C05460=1018.869,-126.788,405.091,165.310,52.720,159.347
C05461=1018.864,-127.038,405.098,165.308,52.725,159.348
C05462=1018.858,-127.287,405.106,165.304,52.729,159.348
C05463=1018.854,-127.537,405.114,165.302,52.734,159.348
C05464=1018.848,-127.787,405.121,165.298,52.738,159.348
C05465=1018.843,-128.036,405.128,165.296,52.743,159.348
C05466=1018.839,-128.285,405.136,165.292,52.747,159.348
C05467=1018.834,-128.535,405.145,165.289,52.751,159.348
C05468=1018.830,-128.785,405.154,165.287,52.754,159.349
C05469=1018.827,-129.034,405.163,165.284,52.757,159.348
C05470=1018.824,-129.284,405.174,165.281,52.759,159.348
C05471=1018.821,-129.534,405.184,165.279,52.761,159.348
C05472=1018.819,-129.783,405.196,165.276,52.761,159.348
C05473=1018.817,-130.033,405.208,165.274,52.762,159.347
C05474=1018.816,-130.283,405.220,165.272,52.762,159.347
C05475=1018.815,-130.532,405.233,165.269,52.762,159.346
C05476=1018.815,-130.782,405.247,165.267,52.761,159.346
C05477=1018.815,-131.032,405.261,165.265,52.759,159.345
C05478=1018.815,-131.282,405.276,165.263,52.757,159.344
C05479=1018.816,-131.532,405.291,165.260,52.754,159.343
C05480=1018.817,-131.781,405.308,165.258,52.752,159.342
C05481=1018.819,-132.031,405.324,165.257,52.748,159.341
C05482=1018.821,-132.281,405.341,165.255,52.744,159.340
C05483=1018.823,-132.531,405.360,165.253,52.739,159.339
C05484=1018.827,-132.780,405.377,165.251,52.734,159.338
C05485=1018.830,-133.030,405.397,165.249,52.728,159.337
C05486=1018.834,-133.280,405.416,165.248,52.722,159.335
C05487=1018.565,-133.306,405.043,165.205,53.048,159.383
C05488=1018.561,-133.056,405.024,165.208,53.054,159.384
C05489=1018.558,-132.806,405.005,165.209,53.060,159.385
C05490=1018.554,-132.557,404.986,165.211,53.065,159.387
C05491=1018.552,-132.307,404.969,165.212,53.070,159.388
C05492=1018.550,-132.057,404.951,165.214,53.074,159.389
C05493=1018.549,-131.808,404.934,165.217,53.077,159.390
C05494=1018.547,-131.558,404.919,165.218,53.080,159.391
C05495=1018.546,-131.308,404.903,165.220,53.083,159.392
C05496=1018.546,-131.058,404.888,165.222,53.085,159.393
C05497=1018.546,-130.808,404.874,165.225,53.087,159.393
C05498=1018.547,-130.559,404.860,165.227,53.088,159.394
C05499=1018.547,-130.309,404.847,165.229,53.088,159.395
C05500=1018.549,-130.059,404.835,165.232,53.088,159.395
C05501=1018.550,-129.810,404.823,165.234,53.087,159.395
C05502=1018.552,-129.560,404.811,165.236,53.087,159.396
C05503=1018.555,-129.311,404.801,165.239,53.085,159.396
C05504=1018.558,-129.060,404.791,165.242,53.083,159.396
C05505=1018.562,-128.811,404.780,165.245,53.080,159.396
C05506=1018.566,-128.562,404.772,165.248,53.077,159.396
C05507=1018.569,-128.312,404.764,165.251,53.073,159.396
C05508=1018.574,-128.062,404.755,165.253,53.069,159.396
C05509=1018.580,-127.813,404.748,165.257,53.064,159.396
C05510=1018.584,-127.563,404.741,165.259,53.059,159.396
C05511=1018.590,-127.314,404.733,165.262,53.054,159.395
C05512=1018.595,-127.064,404.725,165.265,53.050,159.395
C05513=1018.600,-126.814,404.719,165.268,53.045,159.395
C05514=1018.605,-126.564,404.711,165.271,53.041,159.395
C05515=1018.611,-126.314,404.704,165.274,53.036,159.395
C05516=1018.615,-126.064,404.696,165.277,53.031,159.394
C05517=1018.621,-125.814,404.689,165.280,53.026,159.394
C05518=1018.625,-125.565,404.682,165.283,53.021,159.394
C05519=1018.631,-125.315,404.674,165.287,53.017,159.394
C05520=1018.636,-125.065,404.666,165.289,53.012,159.393
C05521=1018.641,-124.816,404.659,165.292,53.007,159.393
C05522=1018.646,-124.565,404.651,165.295,53.003,159.393
C05523=1018.652,-124.315,404.644,165.298,52.998,159.393
C05524=1018.656,-124.066,404.636,165.301,52.994,159.393
C05525=1018.661,-123.816,404.628,165.304,52.989,159.393
C05526=1018.667,-123.566,404.621,165.307,52.983,159.392
C05527=1018.672,-123.317,404.613,165.310,52.979,159.392
C05528=1018.677,-123.067,404.605,165.313,52.974,159.392
C05529=1018.682,-122.817,404.598,165.316,52.970,159.392
C05530=1018.687,-122.566,404.590,165.319,52.965,159.392
C05531=1018.692,-122.317,404.582,165.323,52.961,159.392
C05532=1018.698,-122.067,404.575,165.325,52.956,159.391
C05533=1018.703,-121.817,404.567,165.328,52.951,159.391
C05534=1018.707,-121.568,404.559,165.331,52.947,159.391
C05535=1018.713,-121.318,404.552,165.334,52.942,159.391
C05536=1018.718,-121.068,404.544,165.337,52.938,159.390
C05537=1018.723,-120.818,404.536,165.340,52.933,159.390
C05538=1018.728,-120.569,404.529,165.343,52.927,159.390
C05539=1018.734,-120.319,404.520,165.346,52.923,159.390
C05540=1018.739,-120.068,404.513,165.349,52.918,159.390
C05541=1018.744,-119.818,404.506,165.352,52.914,159.389
C05542=1018.749,-119.569,404.497,165.355,52.909,159.389
C05543=1018.754,-119.319,404.490,165.358,52.904,159.389
C05544=1018.759,-119.069,404.481,165.361,52.900,159.389
C05545=1018.765,-118.819,404.474,165.364,52.895,159.389
C05546=1018.770,-118.570,404.465,165.367,52.891,159.388
C05547=1018.774,-118.320,404.458,165.370,52.886,159.388
C05548=1018.781,-118.036,404.450,165.373,52.881,159.388
C05549=1018.786,-117.752,404.440,165.377,52.875,159.388
C05550=1018.793,-117.468,404.432,165.381,52.869,159.387
C05551=1018.798,-117.184,404.423,165.384,52.865,159.387
C05552=1018.804,-116.934,404.414,165.386,52.860,159.387
C05553=1018.809,-116.684,404.406,165.390,52.855,159.387
C05554=1018.814,-116.435,404.399,165.393,52.850,159.387
C05555=1018.819,-116.186,404.390,165.396,52.846,159.386
C05556=1018.824,-115.935,404.383,165.399,52.841,159.386
C05557=1018.830,-115.685,404.374,165.401,52.836,159.386
C05558=1018.835,-115.435,404.367,165.405,52.832,159.386
C05559=1018.841,-115.186,404.358,165.408,52.827,159.386
C05560=1018.846,-114.935,404.351,165.411,52.823,159.385
C05561=1018.850,-114.686,404.343,165.414,52.818,159.385
C05562=1018.855,-114.437,404.334,165.416,52.813,159.385
C05563=1018.861,-114.187,404.327,165.420,52.808,159.385
C05564=1018.866,-113.937,404.318,165.424,52.803,159.385
C05565=1018.872,-113.687,404.310,165.426,52.799,159.384
C05566=1018.877,-113.437,404.302,165.430,52.794,159.384
C05567=1018.882,-113.187,404.294,165.432,52.790,159.384
C05568=1018.887,-112.937,404.285,165.436,52.785,159.384
C05569=1018.892,-112.687,404.277,165.439,52.780,159.384
C05570=1018.897,-112.437,404.269,165.441,52.776,159.383
C05571=1018.902,-112.188,404.261,165.445,52.771,159.383
C05572=1018.908,-111.939,404.253,165.447,52.767,159.383
C05573=1018.913,-111.689,404.245,165.451,52.762,159.383
C05574=1018.918,-111.439,404.237,165.453,52.758,159.383
C05575=1018.924,-111.189,404.228,165.456,52.752,159.382
C05576=1018.929,-110.940,404.220,165.460,52.748,159.382
C05577=1018.934,-110.689,404.212,165.462,52.743,159.382
C05578=1018.939,-110.439,404.203,165.466,52.739,159.382
C05579=1018.944,-110.190,404.195,165.468,52.734,159.381
C05580=1018.950,-109.940,404.186,165.471,52.729,159.381
///RCONF 1,0,0,0,0,0,0,0,0,0,0,0,0,0,0,0,0,0,0,0,0,0,0,0
C05581=1018.955,-109.690,404.179,165.475,52.724,159.381
C05582=1018.961,-109.440,404.171,165.477,52.720,159.381
C05583=1018.966,-109.191,404.162,165.481,52.715,159.381
C05584=1018.971,-108.941,404.154,165.484,52.711,159.381
C05585=1018.976,-108.691,404.145,165.486,52.706,159.380
C05586=1018.982,-108.441,404.137,165.490,52.701,159.380
C05587=1018.987,-108.191,404.129,165.492,52.697,159.380
C05588=1018.992,-107.941,404.121,165.496,52.692,159.380
C05589=1018.997,-107.692,404.112,165.500,52.687,159.379
C05590=1019.002,-107.442,404.104,165.502,52.682,159.379
C05591=1019.008,-107.192,404.095,165.505,52.678,159.379
C05592=1019.013,-106.943,404.087,165.508,52.673,159.379
C05593=1019.018,-106.693,404.078,165.511,52.669,159.379
C05594=1019.023,-106.443,404.070,165.514,52.664,159.378
C05595=1019.029,-106.193,404.061,165.517,52.660,159.378
C05596=1019.035,-105.943,404.052,165.521,52.655,159.378
C05597=1019.040,-105.693,404.044,165.523,52.650,159.378
C05598=1019.045,-105.444,404.035,165.526,52.645,159.377
C05599=1019.050,-105.194,404.027,165.529,52.641,159.377
C05600=1019.056,-104.944,404.018,165.532,52.636,159.377
C05601=1019.060,-104.694,404.009,165.535,52.632,159.377
C05602=1019.065,-104.444,404.001,165.538,52.627,159.377
C05603=1019.071,-104.195,403.992,165.542,52.623,159.377
C05604=1019.076,-103.945,403.984,165.544,52.618,159.376
C05605=1019.081,-103.695,403.975,165.547,52.613,159.376
C05606=1019.087,-103.445,403.967,165.550,52.609,159.376
C05607=1019.092,-103.195,403.958,165.553,52.604,159.376
C05608=1019.098,-102.945,403.950,165.557,52.599,159.376
C05609=1019.103,-102.696,403.941,165.559,52.595,159.375
C05610=1019.108,-102.446,403.933,165.563,52.590,159.375
C05611=1019.113,-102.197,403.923,165.565,52.585,159.375
C05612=1019.119,-101.912,403.913,165.570,52.580,159.375
C05613=1019.125,-101.628,403.903,165.573,52.575,159.374
C05614=1019.131,-101.345,403.893,165.576,52.570,159.374
C05615=1019.138,-101.060,403.883,165.579,52.564,159.374
C05616=1019.143,-100.811,403.875,165.583,52.560,159.374
C05617=1019.148,-100.561,403.866,165.585,52.555,159.373
C05618=1019.153,-100.311,403.858,165.589,52.551,159.373
C05619=1019.159,-100.061,403.849,165.592,52.546,159.373
C05620=1019.164,-99.811,403.839,165.594,52.541,159.373
C05621=1019.169,-99.562,403.831,165.598,52.536,159.372
C05622=1019.175,-99.312,403.822,165.600,52.532,159.372
C05623=1019.180,-99.062,403.814,165.604,52.527,159.372
C05624=1019.186,-98.812,403.804,165.607,52.522,159.372
C05625=1019.191,-98.563,403.796,165.609,52.518,159.371
C05626=1019.197,-98.313,403.787,165.613,52.513,159.371
C05627=1019.202,-98.063,403.779,165.615,52.509,159.371
C05628=1019.207,-97.813,403.769,165.619,52.504,159.371
C05629=1019.213,-97.563,403.760,165.622,52.499,159.371
C05630=1019.218,-97.314,403.751,165.625,52.495,159.371
C05631=1019.223,-97.064,403.742,165.628,52.490,159.370
C05632=1019.229,-96.814,403.733,165.631,52.486,159.370
C05633=1019.233,-96.564,403.724,165.634,52.481,159.370
C05634=1019.239,-96.315,403.715,165.637,52.477,159.370
C05635=1019.244,-96.064,403.705,165.640,52.472,159.369
C05636=1019.249,-95.815,403.696,165.643,52.468,159.369
C05637=1019.255,-95.565,403.687,165.646,52.463,159.369
C05638=1019.259,-95.316,403.678,165.649,52.459,159.369
C05639=1019.265,-95.065,403.669,165.652,52.454,159.369
C05640=1019.270,-94.815,403.660,165.655,52.450,159.368
C05641=1019.275,-94.566,403.651,165.658,52.445,159.368
C05642=1019.281,-94.316,403.642,165.661,52.441,159.368
C05643=1019.286,-94.066,403.632,165.664,52.436,159.368
C05644=1019.291,-93.817,403.623,165.667,52.432,159.368
C05645=1019.297,-93.567,403.613,165.670,52.427,159.368
C05646=1019.302,-93.317,403.605,165.672,52.422,159.367
C05647=1019.308,-93.068,403.596,165.676,52.418,159.367
C05648=1019.313,-92.817,403.586,165.680,52.413,159.367
C05649=1019.318,-92.568,403.577,165.682,52.409,159.367
C05650=1019.323,-92.319,403.567,165.686,52.404,159.366
C05651=1019.329,-92.068,403.558,165.688,52.400,159.366
C05652=1019.334,-91.819,403.548,165.692,52.395,159.366
C05653=1019.339,-91.569,403.540,165.694,52.391,159.366
C05654=1019.345,-91.319,403.530,165.697,52.386,159.365
C05655=1019.350,-91.069,403.521,165.700,52.381,159.365
C05656=1019.356,-90.819,403.512,165.703,52.377,159.365
C05657=1019.361,-90.570,403.502,165.707,52.372,159.365
C05658=1019.366,-90.320,403.493,165.709,52.368,159.365
C05659=1019.372,-90.070,403.483,165.713,52.363,159.364
C05660=1019.377,-89.821,403.475,165.715,52.358,159.364
C05661=1019.383,-89.571,403.465,165.719,52.353,159.364
C05662=1019.388,-89.321,403.455,165.721,52.349,159.364
C05663=1019.394,-89.071,403.447,165.725,52.345,159.363
C05664=1019.399,-88.821,403.437,165.728,52.340,159.363
C05665=1019.405,-88.572,403.427,165.730,52.335,159.363
C05666=1019.409,-88.322,403.418,165.734,52.330,159.363
C05667=1019.415,-88.073,403.409,165.736,52.326,159.362
C05668=1019.420,-87.822,403.399,165.740,52.321,159.362
C05669=1019.425,-87.573,403.390,165.743,52.317,159.362
C05670=1019.432,-87.323,403.381,165.745,52.312,159.362
C05671=1019.436,-87.074,403.371,165.749,52.307,159.362
C05672=1019.443,-86.824,403.361,165.752,52.303,159.361
C05673=1019.447,-86.574,403.352,165.755,52.298,159.361
C05674=1019.453,-86.324,403.343,165.758,52.293,159.361
C05675=1019.458,-86.075,403.333,165.761,52.289,159.361
C05676=1019.465,-85.792,403.323,165.764,52.283,159.360
C05677=1019.471,-85.510,403.312,165.768,52.278,159.360
C05678=1019.477,-85.229,403.301,165.772,52.273,159.360
C05679=1019.483,-84.947,403.290,165.775,52.268,159.360
C05680=1019.489,-84.697,403.281,165.778,52.262,159.359
C05681=1019.494,-84.447,403.271,165.780,52.258,159.359
C05682=1019.500,-84.198,403.262,165.784,52.253,159.359
C05683=1019.505,-83.948,403.252,165.787,52.249,159.359
C05684=1019.511,-83.698,403.242,165.790,52.244,159.358
C05685=1019.516,-83.448,403.233,165.793,52.239,159.358
C05686=1019.522,-83.199,403.224,165.796,52.235,159.358
C05687=1019.528,-82.949,403.214,165.799,52.230,159.357
C05688=1019.533,-82.699,403.204,165.802,52.225,159.357
C05689=1019.539,-82.450,403.195,165.805,52.221,159.357
C05690=1019.544,-82.199,403.185,165.808,52.215,159.357
C05691=1019.550,-81.950,403.176,165.812,52.211,159.357
C05692=1019.555,-81.700,403.166,165.814,52.207,159.356
C05693=1019.561,-81.451,403.157,165.817,52.201,159.356
C05694=1019.566,-81.200,403.147,165.821,52.197,159.356
C05695=1019.572,-80.951,403.137,165.823,52.192,159.355
C05696=1019.577,-80.701,403.127,165.826,52.187,159.355
C05697=1019.583,-80.451,403.118,165.830,52.182,159.355
C05698=1019.589,-80.201,403.108,165.832,52.177,159.355
C05699=1019.594,-79.952,403.098,165.836,52.173,159.354
C05700=1019.600,-79.702,403.088,165.838,52.169,159.354
C05701=1019.605,-79.452,403.078,165.842,52.164,159.354
C05702=1019.610,-79.203,403.068,165.844,52.160,159.354
C05703=1019.616,-78.953,403.059,165.847,52.154,159.353
C05704=1019.621,-78.703,403.049,165.851,52.150,159.353
C05705=1019.626,-78.453,403.039,165.853,52.145,159.353
C05706=1019.632,-78.203,403.029,165.857,52.141,159.353
C05707=1019.638,-77.955,403.019,165.859,52.137,159.353
C05708=1019.643,-77.705,403.009,165.863,52.131,159.352
C05709=1019.648,-77.454,402.998,165.865,52.127,159.352
C05710=1019.654,-77.204,402.988,165.869,52.122,159.352
C05711=1019.659,-76.955,402.979,165.871,52.118,159.352
C05712=1019.665,-76.705,402.969,165.874,52.113,159.351
C05713=1019.670,-76.455,402.959,165.878,52.108,159.351
C05714=1019.675,-76.206,402.948,165.880,52.104,159.351
C05715=1019.682,-75.956,402.939,165.884,52.099,159.351
C05716=1019.687,-75.706,402.928,165.886,52.094,159.350
C05717=1019.693,-75.456,402.918,165.890,52.090,159.350
C05718=1019.697,-75.207,402.909,165.893,52.085,159.350
C05719=1019.704,-74.958,402.898,165.895,52.080,159.349
C05720=1019.709,-74.708,402.888,165.899,52.076,159.349
C05721=1019.715,-74.457,402.878,165.901,52.071,159.349
C05722=1019.720,-74.208,402.868,165.905,52.067,159.349
C05723=1019.725,-73.959,402.857,165.907,52.063,159.349
C05724=1019.731,-73.708,402.847,165.911,52.058,159.348
C05725=1019.736,-73.458,402.837,165.913,52.053,159.348
C05726=1019.741,-73.210,402.826,165.917,52.048,159.348
C05727=1019.747,-72.959,402.816,165.919,52.044,159.347
C05728=1019.752,-72.709,402.806,165.923,52.040,159.347
C05729=1019.758,-72.460,402.795,165.925,52.035,159.347
C05730=1019.763,-72.210,402.785,165.929,52.031,159.347
C05731=1019.768,-71.961,402.775,165.931,52.027,159.347
C05732=1019.774,-71.711,402.764,165.935,52.022,159.346
C05733=1019.780,-71.461,402.753,165.937,52.017,159.346
C05734=1019.785,-71.211,402.743,165.941,52.012,159.346
C05735=1019.790,-70.961,402.733,165.943,52.008,159.346
C05736=1019.796,-70.712,402.723,165.947,52.004,159.345
C05737=1019.800,-70.462,402.712,165.949,51.999,159.345
C05738=1019.806,-70.212,402.701,165.953,51.995,159.345
C05739=1019.812,-69.962,402.691,165.955,51.990,159.345
C05740=1019.818,-69.683,402.679,165.959,51.985,159.344
C05741=1019.824,-69.403,402.667,165.962,51.980,159.344
C05742=1019.830,-69.123,402.656,165.965,51.975,159.344
C05743=1019.837,-68.843,402.644,165.968,51.970,159.344
C05744=1019.842,-68.594,402.633,165.972,51.965,159.343
C05745=1019.847,-68.344,402.623,165.975,51.960,159.343
C05746=1019.853,-68.095,402.612,165.978,51.956,159.343
C05747=1019.858,-67.844,402.602,165.981,51.951,159.343
C05748=1019.864,-67.595,402.591,165.984,51.947,159.342
C05749=1019.869,-67.345,402.581,165.987,51.942,159.342
C05750=1019.875,-67.095,402.570,165.989,51.937,159.342
C05751=1019.880,-66.846,402.559,165.993,51.933,159.342
C05752=1019.886,-66.595,402.548,165.996,51.929,159.341
C05753=1019.891,-66.347,402.538,165.999,51.923,159.341
C05754=1019.896,-66.097,402.528,166.001,51.919,159.341
C05755=1019.902,-65.847,402.517,166.005,51.915,159.340
C05756=1019.908,-65.598,402.506,166.007,51.910,159.340
C05757=1019.913,-65.347,402.496,166.011,51.905,159.340
C05758=1019.919,-65.098,402.485,166.014,51.900,159.340
C05759=1019.925,-64.848,402.474,166.017,51.896,159.339
C05760=1019.930,-64.598,402.464,166.020,51.892,159.339
C05761=1019.936,-64.349,402.453,166.022,51.887,159.339
C05762=1019.941,-64.099,402.443,166.026,51.882,159.339
C05763=1019.947,-63.849,402.432,166.028,51.878,159.338
C05764=1019.952,-63.599,402.421,166.032,51.873,159.338
C05765=1019.958,-63.350,402.410,166.034,51.868,159.338
C05766=1019.963,-63.100,402.400,166.038,51.864,159.338
C05767=1019.969,-62.850,402.389,166.041,51.858,159.337
C05768=1019.975,-62.601,402.378,166.043,51.854,159.337
C05769=1019.980,-62.351,402.368,166.047,51.850,159.337
C05770=1019.986,-62.101,402.357,166.049,51.845,159.336
C05771=1019.991,-61.852,402.346,166.053,51.840,159.336
C05772=1019.997,-61.602,402.335,166.055,51.836,159.336
C05773=1020.003,-61.352,402.325,166.058,51.831,159.335
C05774=1020.008,-61.103,402.314,166.061,51.826,159.335
C05775=1020.013,-60.853,402.302,166.064,51.822,159.335
C05776=1020.019,-60.603,402.292,166.068,51.817,159.335
C05777=1020.025,-60.353,402.281,166.070,51.812,159.334
C05778=1020.030,-60.104,402.271,166.073,51.807,159.334
C05779=1020.036,-59.854,402.260,166.076,51.803,159.334
C05780=1020.042,-59.604,402.248,166.079,51.798,159.334
C05781=1020.048,-59.355,402.238,166.083,51.793,159.333
C05782=1020.054,-59.105,402.227,166.085,51.789,159.333
C05783=1020.059,-58.855,402.217,166.088,51.783,159.333
C05784=1020.065,-58.606,402.206,166.091,51.779,159.332
C05785=1020.070,-58.356,402.194,166.094,51.774,159.332
C05786=1020.076,-58.106,402.183,166.098,51.769,159.332
C05787=1020.082,-57.857,402.172,166.100,51.765,159.331
C05788=1020.087,-57.607,402.162,166.103,51.760,159.331
C05789=1020.093,-57.357,402.151,166.106,51.756,159.331
C05790=1020.099,-57.107,402.140,166.109,51.750,159.330
C05791=1020.105,-56.857,402.129,166.113,51.746,159.330
C05792=1020.110,-56.608,402.118,166.115,51.741,159.330
C05793=1020.116,-56.358,402.108,166.118,51.736,159.330
C05794=1020.121,-56.109,402.096,166.120,51.731,159.329
C05795=1020.127,-55.859,402.085,166.124,51.727,159.329
C05796=1020.133,-55.610,402.074,166.127,51.722,159.329
C05797=1020.139,-55.360,402.063,166.130,51.717,159.328
C05798=1020.144,-55.109,402.053,166.133,51.712,159.328
C05799=1020.150,-54.860,402.042,166.136,51.708,159.328
C05800=1020.156,-54.610,402.031,166.139,51.703,159.327
C05801=1020.162,-54.361,402.020,166.142,51.698,159.327
C05802=1020.167,-54.110,402.008,166.144,51.693,159.327
C05803=1020.173,-53.861,401.998,166.148,51.689,159.326
C05804=1020.180,-53.582,401.985,166.151,51.683,159.326
C05805=1020.186,-53.304,401.973,166.154,51.678,159.326
C05806=1020.193,-53.025,401.961,166.158,51.673,159.325
C05807=1020.199,-52.746,401.948,166.161,51.667,159.325
C05808=1020.205,-52.497,401.937,166.164,51.662,159.325
C05809=1020.211,-52.247,401.926,166.167,51.657,159.324
C05810=1020.216,-51.998,401.916,166.170,51.653,159.324
C05811=1020.223,-51.748,401.904,166.173,51.648,159.324
C05812=1020.228,-51.498,401.893,166.176,51.643,159.323
C05813=1020.233,-51.248,401.882,166.179,51.638,159.323
C05814=1020.239,-50.999,401.871,166.182,51.633,159.323
C05815=1020.245,-50.749,401.860,166.184,51.629,159.322
C05816=1020.251,-50.500,401.848,166.188,51.624,159.322
C05817=1020.257,-50.250,401.837,166.190,51.619,159.322
C05818=1020.262,-50.000,401.825,166.194,51.615,159.322
C05819=1020.268,-49.750,401.814,166.196,51.610,159.321
C05820=1020.273,-49.501,401.802,166.200,51.606,159.321
C05821=1020.279,-49.251,401.791,166.202,51.601,159.321
C05822=1020.285,-49.001,401.779,166.205,51.596,159.320
C05823=1020.290,-48.752,401.767,166.208,51.592,159.320
C05824=1020.296,-48.502,401.756,166.211,51.587,159.320
C05825=1020.301,-48.252,401.745,166.214,51.583,159.319
C05826=1020.307,-48.002,401.733,166.217,51.577,159.319
C05827=1020.312,-47.753,401.721,166.219,51.573,159.319
C05828=1020.318,-47.504,401.710,166.223,51.569,159.319
C05829=1020.324,-47.253,401.698,166.225,51.564,159.318
C05830=1020.330,-47.004,401.687,166.229,51.559,159.318
C05831=1020.335,-46.754,401.675,166.231,51.555,159.318
C05832=1020.341,-46.505,401.663,166.235,51.550,159.317
C05833=1020.346,-46.255,401.652,166.237,51.546,159.317
C05834=1020.352,-46.006,401.641,166.240,51.540,159.317
C05835=1020.358,-45.756,401.629,166.244,51.536,159.316
C05836=1020.364,-45.506,401.618,166.246,51.532,159.316
C05837=1020.369,-45.256,401.606,166.250,51.526,159.316
C05838=1020.375,-45.007,401.594,166.252,51.522,159.316
C05839=1020.380,-44.757,401.583,166.255,51.517,159.315
C05840=1020.386,-44.507,401.570,166.258,51.513,159.315
C05841=1020.392,-44.258,401.559,166.261,51.508,159.314
C05842=1020.397,-44.008,401.547,166.264,51.503,159.314
C05843=1020.404,-43.758,401.536,166.267,51.498,159.314
C05844=1020.409,-43.508,401.524,166.269,51.494,159.314
C05845=1020.415,-43.259,401.512,166.273,51.489,159.313
C05846=1020.420,-43.009,401.501,166.275,51.484,159.313
C05847=1020.426,-42.760,401.489,166.279,51.480,159.313
C05848=1020.432,-42.510,401.478,166.281,51.475,159.312
C05849=1020.437,-42.261,401.465,166.285,51.470,159.312
C05850=1020.444,-42.010,401.454,166.287,51.466,159.312
C05851=1020.449,-41.761,401.442,166.290,51.461,159.311
C05852=1020.455,-41.512,401.431,166.294,51.456,159.311
C05853=1020.460,-41.262,401.418,166.296,51.452,159.311
C05854=1020.466,-41.012,401.408,166.299,51.446,159.310
C05855=1020.472,-40.762,401.395,166.302,51.442,159.310
C05856=1020.478,-40.513,401.384,166.305,51.437,159.310
C05857=1020.484,-40.263,401.372,166.307,51.432,159.309
C05858=1020.489,-40.014,401.359,166.311,51.428,159.309
C05859=1020.495,-39.764,401.348,166.313,51.423,159.308
C05860=1020.501,-39.514,401.336,166.317,51.418,159.308
C05861=1020.507,-39.264,401.325,166.319,51.413,159.308
C05862=1020.512,-39.015,401.313,166.322,51.409,159.308
C05863=1020.518,-38.765,401.300,166.325,51.405,159.307
C05864=1020.523,-38.515,401.289,166.328,51.399,159.307
C05865=1020.529,-38.266,401.276,166.331,51.395,159.307
C05866=1020.535,-38.017,401.264,166.334,51.390,159.306
C05867=1020.541,-37.767,401.252,166.336,51.386,159.306
C05868=1020.547,-37.488,401.239,166.340,51.380,159.306
C05869=1020.553,-37.210,401.225,166.343,51.375,159.305
C05870=1020.559,-36.932,401.212,166.346,51.370,159.305
C05871=1020.566,-36.653,401.199,166.349,51.365,159.304
C05872=1020.572,-36.403,401.186,166.353,51.360,159.304
C05873=1020.577,-36.154,401.174,166.355,51.355,159.304
C05874=1020.583,-35.904,401.161,166.359,51.351,159.304
C05875=1020.588,-35.654,401.150,166.361,51.347,159.303
C05876=1020.595,-35.405,401.138,166.364,51.341,159.303
C05877=1020.600,-35.156,401.126,166.367,51.337,159.303
C05878=1020.606,-34.906,401.113,166.369,51.332,159.302
C05879=1020.612,-34.656,401.101,166.373,51.328,159.302
C05880=1020.617,-34.406,401.089,166.375,51.323,159.301
C05881=1020.623,-34.156,401.076,166.378,51.318,159.301
C05882=1020.629,-33.907,401.065,166.381,51.314,159.301
C05883=1020.635,-33.657,401.052,166.384,51.309,159.301
C05884=1020.640,-33.408,401.040,166.386,51.304,159.300
C05885=1020.646,-33.158,401.028,166.390,51.300,159.300
C05886=1020.652,-32.909,401.015,166.392,51.295,159.299
C05887=1020.657,-32.659,401.004,166.396,51.290,159.299
C05888=1020.663,-32.409,400.992,166.398,51.285,159.299
C05889=1020.669,-32.160,400.979,166.402,51.281,159.299
C05890=1020.675,-31.910,400.967,166.404,51.276,159.298
C05891=1020.681,-31.660,400.954,166.407,51.272,159.298
C05892=1020.686,-31.411,400.942,166.410,51.267,159.297
C05893=1020.692,-31.161,400.930,166.413,51.262,159.297
C05894=1020.698,-30.911,400.917,166.415,51.257,159.297
C05895=1020.704,-30.662,400.905,166.419,51.252,159.296
C05896=1020.710,-30.413,400.893,166.421,51.248,159.296
C05897=1020.716,-30.163,400.880,166.424,51.243,159.296
C05898=1020.721,-29.913,400.868,166.427,51.239,159.295
C05899=1020.727,-29.664,400.856,166.430,51.233,159.295
C05900=1020.733,-29.414,400.843,166.433,51.229,159.295
C05901=1020.738,-29.165,400.831,166.436,51.224,159.294
C05902=1020.745,-28.915,400.819,166.438,51.219,159.294
C05903=1020.751,-28.665,400.806,166.442,51.215,159.294
C05904=1020.756,-28.416,400.794,166.444,51.210,159.293
C05905=1020.762,-28.166,400.782,166.448,51.205,159.293
C05906=1020.768,-27.916,400.769,166.450,51.200,159.292
C05907=1020.774,-27.666,400.756,166.453,51.195,159.292
C05908=1020.779,-27.417,400.744,166.455,51.191,159.292
C05909=1020.785,-27.167,400.732,166.459,51.186,159.291
C05910=1020.791,-26.917,400.719,166.461,51.182,159.291
C05911=1020.797,-26.667,400.707,166.464,51.176,159.291
C05912=1020.802,-26.418,400.694,166.467,51.172,159.290
C05913=1020.808,-26.168,400.682,166.471,51.168,159.290
C05914=1020.813,-25.919,400.668,166.473,51.163,159.290
C05915=1020.819,-25.670,400.656,166.475,51.159,159.289
C05916=1020.825,-25.420,400.643,166.479,51.153,159.289
C05917=1020.830,-25.170,400.631,166.481,51.149,159.289
C05918=1020.836,-24.920,400.618,166.484,51.144,159.288
C05919=1020.842,-24.671,400.605,166.487,51.140,159.288
C05920=1020.848,-24.421,400.593,166.490,51.135,159.288
C05921=1020.853,-24.171,400.580,166.493,51.131,159.287
C05922=1020.859,-23.921,400.567,166.495,51.126,159.287
C05923=1020.865,-23.673,400.554,166.499,51.121,159.287
C05924=1020.870,-23.423,400.542,166.501,51.116,159.286
C05925=1020.876,-23.173,400.529,166.504,51.112,159.286
C05926=1020.882,-22.923,400.516,166.507,51.107,159.285
C05927=1020.889,-22.674,400.503,166.510,51.103,159.285
C05928=1020.893,-22.424,400.490,166.512,51.098,159.285
C05929=1020.899,-22.175,400.478,166.515,51.093,159.284
C05930=1020.905,-21.925,400.465,166.518,51.088,159.284
C05931=1020.911,-21.675,400.452,166.520,51.083,159.284
C05932=1020.918,-21.396,400.438,166.524,51.078,159.283
C05933=1020.924,-21.117,400.423,166.527,51.073,159.283
C05934=1020.930,-20.838,400.409,166.530,51.068,159.282
C05935=1020.936,-20.559,400.395,166.533,51.063,159.282
C05936=1020.942,-20.309,400.382,166.537,51.058,159.282
C05937=1020.948,-20.059,400.369,166.539,51.053,159.281
C05938=1020.954,-19.810,400.356,166.542,51.048,159.281
C05939=1020.961,-19.560,400.343,166.545,51.043,159.280
C05940=1020.967,-19.310,400.331,166.548,51.039,159.280
C05941=1020.971,-19.061,400.318,166.550,51.034,159.280
C05942=1020.977,-18.812,400.304,166.554,51.030,159.280
C05943=1020.983,-18.562,400.292,166.556,51.025,159.279
C05944=1020.989,-18.312,400.279,166.558,51.020,159.279
C05945=1020.995,-18.063,400.266,166.562,51.015,159.278
C05946=1021.001,-17.813,400.254,166.564,51.010,159.278
C05947=1021.007,-17.563,400.240,166.568,51.005,159.277
C05948=1021.013,-17.313,400.227,166.570,51.001,159.277
C05949=1021.019,-17.064,400.214,166.573,50.996,159.277
C05950=1021.024,-16.815,400.202,166.576,50.991,159.276
C05951=1021.030,-16.566,400.188,166.579,50.987,159.276
C05952=1021.036,-16.316,400.176,166.581,50.982,159.276
C05953=1021.041,-16.066,400.163,166.585,50.977,159.275
C05954=1021.048,-15.816,400.149,166.587,50.972,159.275
C05955=1021.054,-15.566,400.137,166.590,50.967,159.275
C05956=1021.059,-15.317,400.123,166.593,50.963,159.274
C05957=1021.065,-15.068,400.110,166.595,50.958,159.274
C05958=1021.070,-14.817,400.097,166.598,50.953,159.273
C05959=1021.077,-14.568,400.083,166.601,50.949,159.273
C05960=1021.083,-14.319,400.070,166.603,50.944,159.272
C05961=1021.088,-14.069,400.057,166.607,50.940,159.272
C05962=1021.094,-13.819,400.044,166.609,50.935,159.272
C05963=1021.099,-13.569,400.031,166.613,50.930,159.272
C05964=1021.106,-13.320,400.017,166.615,50.926,159.271
C05965=1021.111,-13.070,400.003,166.618,50.921,159.271
C05966=1021.116,-12.821,399.991,166.621,50.916,159.270
C05967=1021.123,-12.572,399.978,166.623,50.912,159.270
C05968=1021.128,-12.322,399.964,166.627,50.907,159.270
C05969=1021.134,-12.073,399.951,166.629,50.902,159.269
C05970=1021.139,-11.823,399.938,166.631,50.898,159.269
C05971=1021.146,-11.574,399.924,166.635,50.893,159.268
C05972=1021.151,-11.324,399.910,166.637,50.889,159.268
C05973=1021.157,-11.074,399.898,166.640,50.883,159.268
C05974=1021.163,-10.825,399.884,166.643,50.879,159.267
C05975=1021.169,-10.575,399.871,166.645,50.875,159.267
C05976=1021.175,-10.326,399.858,166.649,50.869,159.267
C05977=1021.180,-10.076,399.844,166.651,50.865,159.266
C05978=1021.186,-9.827,399.831,166.654,50.860,159.266
C05979=1021.192,-9.577,399.817,166.657,50.855,159.265
C05980=1021.199,-9.327,399.804,166.659,50.850,159.265
C05981=1021.204,-9.077,399.790,166.662,50.846,159.265
C05982=1021.210,-8.828,399.777,166.665,50.841,159.264
C05983=1021.216,-8.578,399.763,166.668,50.836,159.264
C05984=1021.222,-8.329,399.750,166.671,50.832,159.263
C05985=1021.227,-8.079,399.736,166.674,50.827,159.263
C05986=1021.233,-7.829,399.724,166.676,50.822,159.263
C05987=1021.239,-7.580,399.710,166.679,50.818,159.262
C05988=1021.245,-7.330,399.697,166.682,50.813,159.262
C05989=1021.251,-7.081,399.683,166.684,50.808,159.261
C05990=1021.257,-6.832,399.669,166.688,50.803,159.261
C05991=1021.262,-6.582,399.657,166.690,50.798,159.261
C05992=1021.268,-6.332,399.643,166.693,50.793,159.260
C05993=1021.274,-6.083,399.630,166.695,50.788,159.260
C05994=1021.280,-5.833,399.615,166.698,50.784,159.259
C05995=1021.286,-5.583,399.602,166.701,50.779,159.259
C05996=1021.293,-5.303,399.587,166.704,50.774,159.259
C05997=1021.299,-5.021,399.572,166.707,50.768,159.258
C05998=1021.306,-4.741,399.556,166.711,50.763,159.258
C05999=1021.312,-4.459,399.541,166.714,50.758,159.257
C06000=1021.318,-4.210,399.528,166.716,50.753,159.257
C06001=1021.324,-3.960,399.514,166.719,50.748,159.256
C06002=1021.329,-3.711,399.500,166.722,50.744,159.256
C06003=1021.336,-3.461,399.487,166.724,50.739,159.255
C06004=1021.342,-3.211,399.473,166.727,50.735,159.255
C06005=1021.348,-2.962,399.458,166.730,50.730,159.255
C06006=1021.353,-2.713,399.444,166.733,50.726,159.254
C06007=1021.358,-2.463,399.431,166.735,50.721,159.254
C06008=1021.364,-2.213,399.417,166.739,50.716,159.254
C06009=1021.370,-1.964,399.403,166.741,50.711,159.253
C06010=1021.376,-1.714,399.389,166.743,50.707,159.253
C06011=1021.382,-1.464,399.375,166.747,50.702,159.253
C06012=1021.387,-1.215,399.362,166.749,50.697,159.252
C06013=1021.393,-0.966,399.347,166.751,50.693,159.252
C06014=1021.398,-0.716,399.333,166.755,50.688,159.251
C06015=1021.405,-0.467,399.320,166.757,50.683,159.251
C06016=1021.411,-0.217,399.306,166.760,50.679,159.250
C06017=1021.416,0.033,399.292,166.763,50.674,159.250
C06018=1021.422,0.282,399.278,166.765,50.670,159.250
C06019=1021.427,0.531,399.263,166.768,50.665,159.249
C06020=1021.434,0.781,399.250,166.771,50.660,159.249
C06021=1021.439,1.030,399.236,166.774,50.656,159.249
C06022=1021.445,1.281,399.222,166.776,50.651,159.248
C06023=1021.451,1.530,399.208,166.779,50.646,159.248
C06024=1021.457,1.779,399.193,166.782,50.642,159.247
C06025=1021.462,2.029,399.180,166.784,50.637,159.247
C06026=1021.468,2.279,399.165,166.788,50.633,159.247
C06027=1021.474,2.528,399.152,166.790,50.628,159.246
C06028=1021.480,2.778,399.138,166.792,50.623,159.246
C06029=1021.486,3.027,399.124,166.796,50.619,159.245
C06030=1021.492,3.277,399.109,166.798,50.614,159.245
C06031=1021.497,3.527,399.096,166.800,50.609,159.244
C06032=1021.503,3.776,399.081,166.803,50.604,159.244
C06033=1021.509,4.025,399.068,166.806,50.600,159.244
C06034=1021.515,4.275,399.053,166.809,50.595,159.243
C06035=1021.521,4.525,399.040,166.811,50.590,159.243
C06036=1021.526,4.774,399.025,166.814,50.586,159.242
C06037=1021.532,5.023,399.011,166.817,50.581,159.242
C06038=1021.538,5.273,398.997,166.820,50.576,159.241
C06039=1021.544,5.522,398.983,166.822,50.571,159.241
C06040=1021.550,5.772,398.969,166.826,50.567,159.241
C06041=1021.556,6.022,398.955,166.828,50.562,159.240
C06042=1021.562,6.271,398.940,166.830,50.557,159.240
C06043=1021.567,6.520,398.926,166.833,50.552,159.239
C06044=1021.573,6.770,398.913,166.836,50.548,159.239
C06045=1021.579,7.020,398.898,166.838,50.543,159.238
C06046=1021.585,7.269,398.884,166.841,50.538,159.238
C06047=1021.591,7.519,398.870,166.844,50.533,159.238
C06048=1021.597,7.768,398.856,166.847,50.529,159.237
C06049=1021.603,8.018,398.842,166.850,50.524,159.237
C06050=1021.608,8.267,398.827,166.852,50.519,159.236
C06051=1021.615,8.517,398.813,166.855,50.514,159.236
C06052=1021.620,8.767,398.799,166.857,50.509,159.235
C06053=1021.627,9.016,398.785,166.860,50.505,159.235
C06054=1021.633,9.266,398.771,166.863,50.500,159.235
C06055=1021.638,9.514,398.756,166.865,50.495,159.234
C06056=1021.644,9.781,398.741,166.869,50.490,159.234
C06057=1021.651,10.048,398.726,166.872,50.485,159.233
C06058=1021.658,10.314,398.711,166.874,50.479,159.233
C06059=1021.664,10.580,398.695,166.877,50.474,159.232
C06060=1021.670,10.845,398.680,166.880,50.469,159.232
C06061=1021.676,11.112,398.665,166.883,50.464,159.231
C06062=1021.683,11.378,398.650,166.886,50.459,159.231
C06063=1021.689,11.644,398.635,166.889,50.454,159.231
C06064=1021.695,11.893,398.620,166.891,50.449,159.230
C06065=1021.701,12.144,398.606,166.894,50.445,159.229
C06066=1021.707,12.393,398.591,166.897,50.439,159.229
C06067=1021.713,12.643,398.577,166.899,50.435,159.229
C06068=1021.719,12.892,398.563,166.903,50.429,159.228
C06069=1021.725,13.142,398.548,166.905,50.425,159.228
C06070=1021.731,13.391,398.534,166.907,50.420,159.227
C06071=1021.736,13.641,398.520,166.911,50.416,159.227
C06072=1021.743,13.890,398.505,166.913,50.411,159.226
C06073=1021.748,14.139,398.490,166.915,50.406,159.226
C06074=1021.754,14.390,398.476,166.919,50.401,159.225
C06075=1021.760,14.638,398.462,166.921,50.397,159.225
C06076=1021.767,14.888,398.447,166.923,50.392,159.225
C06077=1021.771,15.138,398.432,166.927,50.387,159.224
C06078=1021.777,15.387,398.418,166.929,50.382,159.224
C06079=1021.784,15.637,398.403,166.932,50.378,159.223
C06080=1021.789,15.886,398.389,166.935,50.373,159.223
C06081=1021.795,16.136,398.374,166.937,50.368,159.222
C06082=1021.801,16.385,398.359,166.939,50.363,159.222
C06083=1021.807,16.635,398.344,166.943,50.359,159.222
C06084=1021.812,16.884,398.330,166.945,50.354,159.221
C06085=1021.819,17.134,398.315,166.948,50.349,159.221
C06086=1021.824,17.383,398.300,166.951,50.344,159.220
C06087=1021.831,17.633,398.285,166.953,50.340,159.220
C06088=1021.836,17.882,398.272,166.956,50.335,159.219
C06089=1021.843,18.132,398.257,166.958,50.331,159.219
C06090=1021.848,18.381,398.241,166.961,50.326,159.219
C06091=1021.854,18.631,398.227,166.964,50.321,159.218
C06092=1021.860,18.880,398.213,166.966,50.316,159.217
C06093=1021.866,19.130,398.198,166.969,50.311,159.217
C06094=1021.872,19.379,398.183,166.972,50.307,159.217
C06095=1021.877,19.629,398.168,166.974,50.302,159.216
C06096=1021.883,19.878,398.153,166.977,50.297,159.216
C06097=1021.890,20.128,398.138,166.980,50.292,159.215
C06098=1021.894,20.377,398.124,166.982,50.288,159.215
C06099=1021.901,20.627,398.109,166.986,50.283,159.215
C06100=1021.906,20.876,398.094,166.988,50.278,159.214
C06101=1021.912,21.126,398.079,166.990,50.274,159.214
C06102=1021.918,21.375,398.064,166.992,50.269,159.213
C06103=1021.924,21.625,398.049,166.996,50.264,159.213
C06104=1021.931,21.874,398.034,166.998,50.260,159.212
C06105=1021.936,22.124,398.019,167.001,50.255,159.212
C06106=1021.942,22.373,398.004,167.004,50.250,159.211
C06107=1021.948,22.622,397.989,167.006,50.245,159.211
C06108=1021.954,22.872,397.974,167.009,50.241,159.211
C06109=1021.959,23.121,397.959,167.012,50.236,159.210
C06110=1021.966,23.371,397.944,167.014,50.231,159.210
C06111=1021.971,23.621,397.929,167.017,50.226,159.209
C06112=1021.977,23.870,397.914,167.019,50.222,159.209
C06113=1021.984,24.119,397.899,167.022,50.216,159.208
C06114=1021.989,24.369,397.884,167.025,50.212,159.208
C06115=1021.995,24.618,397.869,167.027,50.208,159.207
C06116=1022.001,24.868,397.854,167.030,50.203,159.207
C06117=1022.006,25.117,397.839,167.033,50.198,159.206
C06118=1022.013,25.367,397.824,167.035,50.193,159.206
C06119=1022.019,25.616,397.809,167.038,50.188,159.205
C06120=1022.024,25.866,397.794,167.040,50.183,159.205
C06121=1022.031,26.115,397.779,167.043,50.179,159.205
C06122=1022.036,26.364,397.764,167.046,50.174,159.204
C06123=1022.042,26.614,397.749,167.049,50.169,159.204
C06124=1022.049,26.899,397.732,167.052,50.164,159.203
C06125=1022.055,27.183,397.715,167.055,50.158,159.203
C06126=1022.062,27.467,397.697,167.058,50.153,159.202
C06127=1022.069,27.752,397.680,167.061,50.148,159.202
C06128=1022.074,28.001,397.665,167.063,50.143,159.201
C06129=1022.081,28.251,397.650,167.066,50.138,159.201
C06130=1022.086,28.501,397.634,167.068,50.133,159.200
C06131=1022.092,28.749,397.620,167.072,50.129,159.200
C06132=1022.098,28.999,397.603,167.074,50.124,159.199
C06133=1022.104,29.248,397.589,167.076,50.119,159.199
C06134=1022.109,29.498,397.573,167.079,50.115,159.198
C06135=1022.115,29.748,397.558,167.082,50.110,159.198
C06136=1022.122,29.997,397.542,167.085,50.106,159.198
C06137=1022.127,30.246,397.527,167.087,50.101,159.197
C06138=1022.133,30.496,397.512,167.089,50.096,159.196
C06139=1022.139,30.746,397.496,167.092,50.091,159.196
C06140=1022.145,30.994,397.481,167.095,50.086,159.196
C06141=1022.151,31.244,397.466,167.097,50.082,159.195
C06142=1022.156,31.494,397.450,167.101,50.077,159.195
C06143=1022.162,31.743,397.436,167.103,50.072,159.194
C06144=1022.168,31.992,397.419,167.105,50.068,159.194
C06145=1022.174,32.242,397.404,167.108,50.063,159.193
C06146=1022.180,32.492,397.389,167.111,50.058,159.193
C06147=1022.186,32.740,397.373,167.113,50.053,159.192
C06148=1022.192,32.990,397.358,167.115,50.048,159.192
C06149=1022.197,33.240,397.342,167.118,50.044,159.191
C06150=1022.203,33.489,397.328,167.121,50.039,159.191
C06151=1022.209,33.738,397.312,167.124,50.035,159.190
C06152=1022.215,33.988,397.297,167.126,50.030,159.190
C06153=1022.221,34.238,397.281,167.129,50.025,159.190
C06154=1022.227,34.486,397.266,167.132,50.020,159.189
C06155=1022.233,34.736,397.250,167.134,50.015,159.189
C06156=1022.239,34.986,397.234,167.137,50.010,159.188
C06157=1022.245,35.235,397.219,167.139,50.005,159.188
C06158=1022.250,35.485,397.204,167.142,50.001,159.187
C06159=1022.257,35.734,397.188,167.144,49.996,159.187
C06160=1022.262,35.984,397.173,167.147,49.991,159.186
C06161=1022.268,36.234,397.157,167.150,49.987,159.186
C06162=1022.275,36.483,397.141,167.152,49.982,159.185
C06163=1022.280,36.732,397.126,167.156,49.977,159.185
C06164=1022.286,36.981,397.110,167.158,49.972,159.184
C06165=1022.292,37.231,397.095,167.160,49.968,159.184
C06166=1022.298,37.480,397.079,167.163,49.963,159.183
C06167=1022.304,37.730,397.063,167.166,49.958,159.183
C06168=1022.309,37.979,397.047,167.169,49.954,159.183
C06169=1022.315,38.229,397.032,167.171,49.949,159.182
C06170=1022.321,38.478,397.016,167.173,49.944,159.181
C06171=1022.327,38.728,397.001,167.176,49.939,159.181
C06172=1022.333,38.977,396.984,167.179,49.935,159.181
C06173=1022.338,39.226,396.969,167.181,49.930,159.180
C06174=1022.344,39.476,396.953,167.184,49.926,159.180
C06175=1022.350,39.725,396.937,167.186,49.921,159.179
C06176=1022.356,39.975,396.921,167.189,49.916,159.179
C06177=1022.362,40.224,396.905,167.192,49.911,159.178
C06178=1022.368,40.474,396.890,167.194,49.907,159.178
C06179=1022.373,40.723,396.874,167.196,49.902,159.177
C06180=1022.379,40.972,396.858,167.200,49.897,159.177
C06181=1022.385,41.222,396.842,167.202,49.892,159.176
C06182=1022.391,41.471,396.826,167.205,49.888,159.176
C06183=1022.397,41.721,396.811,167.208,49.883,159.175
C06184=1022.403,41.970,396.795,167.210,49.878,159.175
C06185=1022.409,42.219,396.779,167.212,49.874,159.174
C06186=1022.414,42.469,396.763,167.215,49.869,159.174
C06187=1022.420,42.718,396.747,167.218,49.864,159.173
C06188=1022.427,43.003,396.728,167.220,49.859,159.173
C06189=1022.433,43.287,396.711,167.223,49.853,159.172
C06190=1022.440,43.571,396.693,167.227,49.848,159.172
C06191=1022.447,43.855,396.674,167.230,49.843,159.171
C06192=1022.453,44.105,396.658,167.232,49.839,159.171
C06193=1022.458,44.354,396.641,167.235,49.834,159.170
C06194=1022.463,44.604,396.625,167.237,49.829,159.170
C06195=1022.469,44.854,396.609,167.240,49.825,159.170
C06196=1022.475,45.102,396.593,167.242,49.820,159.169
C06197=1022.481,45.352,396.577,167.245,49.815,159.169
C06198=1022.487,45.601,396.561,167.248,49.811,159.168
C06199=1022.493,45.850,396.544,167.250,49.806,159.168
C06200=1022.498,46.100,396.529,167.253,49.802,159.167
C06201=1022.503,46.350,396.512,167.255,49.797,159.167
C06202=1022.509,46.599,396.496,167.258,49.792,159.166
C06203=1022.515,46.849,396.479,167.261,49.787,159.166
C06204=1022.521,47.098,396.463,167.263,49.783,159.165
C06205=1022.527,47.348,396.447,167.266,49.779,159.165
C06206=1022.533,47.596,396.431,167.268,49.774,159.164
C06207=1022.538,47.846,396.416,167.271,49.769,159.164
C06208=1022.544,48.095,396.399,167.274,49.764,159.163
C06209=1022.549,48.345,396.382,167.276,49.760,159.163
C06210=1022.555,48.594,396.366,167.278,49.755,159.162
C06211=1022.561,48.844,396.350,167.280,49.750,159.162
C06212=1022.567,49.093,396.334,167.284,49.746,159.162
C06213=1022.573,49.343,396.317,167.286,49.741,159.161
C06214=1022.579,49.592,396.301,167.289,49.736,159.161
C06215=1022.585,49.841,396.285,167.291,49.732,159.160
C06216=1022.591,50.091,396.269,167.294,49.727,159.160
C06217=1022.596,50.340,396.252,167.297,49.722,159.159
C06218=1022.602,50.590,396.236,167.299,49.717,159.159
C06219=1022.608,50.839,396.219,167.301,49.713,159.158
C06220=1022.614,51.088,396.203,167.305,49.708,159.158
C06221=1022.620,51.338,396.187,167.307,49.704,159.157
C06222=1022.626,51.587,396.170,167.310,49.699,159.157
C06223=1022.632,51.836,396.154,167.312,49.694,159.156
C06224=1022.637,52.086,396.137,167.314,49.689,159.156
C06225=1022.643,52.335,396.121,167.318,49.684,159.155
C06226=1022.649,52.585,396.105,167.320,49.680,159.155
C06227=1022.655,52.834,396.089,167.322,49.675,159.154
C06228=1022.661,53.083,396.072,167.325,49.670,159.154
C06229=1022.667,53.333,396.056,167.328,49.665,159.153
C06230=1022.673,53.582,396.040,167.330,49.661,159.153
C06231=1022.678,53.832,396.023,167.333,49.656,159.152
C06232=1022.684,54.081,396.007,167.335,49.651,159.152
C06233=1022.690,54.330,395.990,167.338,49.646,159.151
C06234=1022.696,54.580,395.974,167.341,49.641,159.151
C06235=1022.702,54.829,395.958,167.343,49.637,159.150
C06236=1022.708,55.078,395.942,167.346,49.633,159.150
C06237=1022.714,55.328,395.925,167.349,49.628,159.149
C06238=1022.719,55.577,395.909,167.351,49.623,159.149
C06239=1022.725,55.827,395.892,167.354,49.618,159.148
C06240=1022.731,56.076,395.876,167.357,49.613,159.148
C06241=1022.737,56.326,395.859,167.359,49.609,159.147
C06242=1022.744,56.575,395.842,167.362,49.604,159.147
C06243=1022.750,56.824,395.826,167.364,49.599,159.146
C06244=1022.755,57.074,395.809,167.367,49.594,159.146
C06245=1022.761,57.323,395.793,167.370,49.590,159.145
C06246=1022.767,57.573,395.777,167.372,49.585,159.145
C06247=1022.773,57.822,395.761,167.374,49.580,159.144
C06248=1022.779,58.071,395.744,167.377,49.575,159.144
C06249=1022.785,58.320,395.727,167.380,49.570,159.143
C06250=1022.791,58.569,395.711,167.382,49.565,159.143
C06251=1022.797,58.820,395.694,167.386,49.560,159.142
C06252=1022.803,59.104,395.675,167.388,49.555,159.142
C06253=1022.810,59.388,395.657,167.391,49.550,159.141
C06254=1022.817,59.671,395.638,167.394,49.544,159.140
C06255=1022.824,59.956,395.619,167.397,49.538,159.140
C06256=1022.830,60.205,395.603,167.399,49.534,159.139
C06257=1022.836,60.454,395.586,167.403,49.529,159.139
C06258=1022.842,60.704,395.569,167.405,49.524,159.138
C06259=1022.848,60.953,395.553,167.407,49.519,159.138
C06260=1022.854,61.203,395.536,167.411,49.514,159.137
C06261=1022.860,61.452,395.520,167.413,49.510,159.137
C06262=1022.866,61.701,395.503,167.415,49.505,159.136
C06263=1022.872,61.950,395.487,167.419,49.500,159.136
C06264=1022.878,62.201,395.470,167.421,49.495,159.135
C06265=1022.884,62.450,395.453,167.423,49.490,159.135
C06266=1022.890,62.699,395.436,167.425,49.485,159.134
C06267=1022.896,62.948,395.420,167.429,49.480,159.134
C06268=1022.902,63.197,395.404,167.431,49.476,159.133
C06269=1022.908,63.447,395.386,167.433,49.471,159.133
C06270=1022.914,63.696,395.370,167.437,49.466,159.132
C06271=1022.919,63.946,395.353,167.439,49.461,159.132
C06272=1022.925,64.195,395.336,167.441,49.457,159.131
C06273=1022.931,64.444,395.319,167.444,49.452,159.131
C06274=1022.937,64.694,395.302,167.446,49.447,159.130
C06275=1022.943,64.944,395.285,167.449,49.442,159.130
C06276=1022.949,65.193,395.269,167.452,49.438,159.129
C06277=1022.954,65.442,395.251,167.454,49.433,159.129
C06278=1022.960,65.691,395.235,167.457,49.428,159.128
C06279=1022.966,65.941,395.217,167.460,49.423,159.128
C06280=1022.972,66.190,395.201,167.462,49.419,159.127
C06281=1022.978,66.439,395.183,167.465,49.414,159.127
C06282=1022.984,66.689,395.167,167.467,49.409,159.126
C06283=1022.990,66.939,395.149,167.471,49.405,159.126
C06284=1022.996,67.188,395.133,167.473,49.400,159.125
C06285=1023.001,67.437,395.115,167.475,49.396,159.125
C06286=1023.007,67.686,395.099,167.478,49.391,159.124
C06287=1023.013,67.935,395.081,167.481,49.386,159.124
C06288=1023.019,68.185,395.065,167.483,49.381,159.123
C06289=1023.025,68.434,395.047,167.486,49.377,159.123
C06290=1023.030,68.683,395.029,167.488,49.372,159.122
C06291=1023.036,68.933,395.013,167.491,49.367,159.122
C06292=1023.042,69.183,394.995,167.494,49.362,159.121
C06293=1023.048,69.432,394.978,167.496,49.358,159.121
C06294=1023.054,69.681,394.961,167.499,49.353,159.120
C06295=1023.059,69.930,394.944,167.501,49.348,159.120
C06296=1023.065,70.180,394.927,167.504,49.343,159.119
C06297=1023.071,70.429,394.910,167.507,49.339,159.119
C06298=1023.077,70.678,394.892,167.509,49.334,159.118
C06299=1023.082,70.928,394.875,167.511,49.329,159.118
C06300=1023.089,71.177,394.858,167.514,49.325,159.117
C06301=1023.094,71.426,394.840,167.517,49.320,159.117
C06302=1023.100,71.676,394.823,167.519,49.315,159.116
C06303=1023.107,71.925,394.806,167.522,49.310,159.116
C06304=1023.112,72.174,394.789,167.524,49.306,159.115
C06305=1023.117,72.424,394.772,167.528,49.301,159.115
C06306=1023.123,72.673,394.754,167.530,49.297,159.114
C06307=1023.130,72.922,394.737,167.533,49.292,159.114
C06308=1023.135,73.172,394.719,167.535,49.288,159.113
C06309=1023.140,73.421,394.702,167.537,49.283,159.113
C06310=1023.147,73.671,394.685,167.541,49.278,159.112
C06311=1023.153,73.920,394.667,167.543,49.273,159.112
C06312=1023.158,74.169,394.650,167.545,49.269,159.111
C06313=1023.164,74.419,394.633,167.548,49.264,159.111
C06314=1023.170,74.668,394.616,167.551,49.259,159.110
C06315=1023.176,74.917,394.598,167.554,49.254,159.110
C06316=1023.183,75.201,394.578,167.557,49.249,159.109
C06317=1023.189,75.485,394.559,167.560,49.243,159.108
C06318=1023.196,75.769,394.539,167.562,49.238,159.108
C06319=1023.203,76.053,394.519,167.565,49.233,159.107
C06320=1023.208,76.302,394.501,167.568,49.228,159.107
C06321=1023.215,76.551,394.484,167.571,49.223,159.106
C06322=1023.221,76.801,394.466,167.573,49.219,159.106
C06323=1023.226,77.050,394.450,167.576,49.214,159.105
C06324=1023.231,77.299,394.432,167.578,49.209,159.105
C06325=1023.238,77.549,394.414,167.581,49.204,159.104
C06326=1023.243,77.798,394.396,167.584,49.200,159.104
C06327=1023.249,78.048,394.379,167.586,49.195,159.103
C06328=1023.255,78.297,394.361,167.588,49.190,159.103
C06329=1023.260,78.546,394.343,167.591,49.186,159.102
C06330=1023.266,78.796,394.325,167.595,49.181,159.102
C06331=1023.272,79.045,394.308,167.597,49.177,159.101
C06332=1023.277,79.294,394.290,167.599,49.172,159.101
C06333=1023.284,79.543,394.272,167.602,49.168,159.100
C06334=1023.289,79.793,394.255,167.604,49.163,159.100
C06335=1023.295,80.042,394.237,167.607,49.158,159.099
C06336=1023.301,80.291,394.219,167.610,49.153,159.099
C06337=1023.306,80.540,394.202,167.612,49.149,159.098
C06338=1023.312,80.790,394.184,167.615,49.144,159.098
C06339=1023.318,81.039,394.166,167.617,49.139,159.097
C06340=1023.324,81.289,394.148,167.620,49.134,159.097
C06341=1023.330,81.538,394.131,167.623,49.130,159.096
C06342=1023.335,81.787,394.113,167.625,49.125,159.096
C06343=1023.341,82.037,394.095,167.628,49.121,159.095
C06344=1023.347,82.286,394.078,167.631,49.116,159.095
C06345=1023.353,82.535,394.060,167.634,49.112,159.094
C06346=1023.359,82.784,394.042,167.636,49.107,159.094
C06347=1023.365,83.034,394.024,167.638,49.102,159.093
C06348=1023.370,83.283,394.006,167.641,49.098,159.093
C06349=1023.376,83.532,393.988,167.644,49.093,159.092
C06350=1023.382,83.781,393.971,167.647,49.088,159.092
C06351=1023.387,84.030,393.953,167.649,49.084,159.091
C06352=1023.394,84.280,393.935,167.651,49.079,159.091
C06353=1023.399,84.529,393.917,167.655,49.074,159.090
C06354=1023.405,84.779,393.900,167.657,49.069,159.090
C06355=1023.411,85.027,393.881,167.659,49.065,159.089
C06356=1023.417,85.277,393.863,167.662,49.060,159.089
C06357=1023.423,85.526,393.846,167.665,49.055,159.088
C06358=1023.429,85.776,393.828,167.668,49.051,159.088
C06359=1023.434,86.025,393.810,167.670,49.046,159.087
C06360=1023.440,86.275,393.792,167.672,49.041,159.087
C06361=1023.446,86.524,393.775,167.676,49.036,159.086
C06362=1023.452,86.773,393.756,167.678,49.032,159.086
C06363=1023.458,87.022,393.739,167.681,49.027,159.085
C06364=1023.464,87.272,393.721,167.684,49.022,159.085
C06365=1023.469,87.521,393.703,167.686,49.018,159.084
C06366=1023.476,87.770,393.685,167.689,49.013,159.084
C06367=1023.481,88.019,393.667,167.691,49.008,159.083
C06368=1023.488,88.269,393.649,167.694,49.003,159.082
C06369=1023.493,88.518,393.631,167.697,48.998,159.082
C06370=1023.499,88.767,393.613,167.699,48.994,159.081
C06371=1023.505,89.016,393.595,167.701,48.989,159.081
C06372=1023.511,89.266,393.577,167.705,48.984,159.080
C06373=1023.517,89.516,393.559,167.707,48.979,159.080
C06374=1023.522,89.765,393.541,167.710,48.975,159.079
C06375=1023.528,90.014,393.522,167.712,48.971,159.079
C06376=1023.533,90.263,393.504,167.716,48.966,159.078
C06377=1023.540,90.512,393.486,167.718,48.961,159.078
C06378=1023.545,90.761,393.468,167.721,48.957,159.077
C06379=1023.551,91.011,393.450,167.723,48.952,159.077
C06380=1023.557,91.295,393.429,167.726,48.946,159.076
C06381=1023.564,91.579,393.408,167.729,48.942,159.076
C06382=1023.571,91.863,393.387,167.732,48.936,159.075
C06383=1023.577,92.146,393.367,167.735,48.931,159.075
C06384=1023.583,92.396,393.348,167.738,48.926,159.074
C06385=1023.588,92.645,393.330,167.741,48.922,159.074
C06386=1023.595,92.894,393.311,167.743,48.917,159.073
C06387=1023.599,93.143,393.293,167.745,48.913,159.073
C06388=1023.606,93.392,393.275,167.749,48.908,159.072
C06389=1023.612,93.642,393.257,167.751,48.903,159.072
C06390=1023.617,93.891,393.238,167.754,48.898,159.071
C06391=1023.623,94.141,393.220,167.756,48.894,159.071
C06392=1023.629,94.389,393.202,167.760,48.889,159.070
C06393=1023.634,94.639,393.183,167.762,48.884,159.070
C06394=1023.641,94.888,393.164,167.764,48.880,159.069
C06395=1023.646,95.137,393.147,167.767,48.875,159.068
C06396=1023.652,95.387,393.128,167.770,48.870,159.068
C06397=1023.658,95.636,393.110,167.773,48.866,159.067
C06398=1023.664,95.885,393.091,167.775,48.861,159.067
C06399=1023.669,96.135,393.073,167.777,48.856,159.066
C06400=1023.675,96.383,393.055,167.781,48.851,159.066
C06401=1023.681,96.633,393.037,167.783,48.847,159.065
C06402=1023.687,96.883,393.017,167.786,48.842,159.065
C06403=1023.692,97.132,393.000,167.788,48.838,159.064
C06404=1023.699,97.381,392.981,167.791,48.833,159.064
C06405=1023.705,97.630,392.962,167.794,48.828,159.063
C06406=1023.710,97.879,392.944,167.796,48.824,159.063
C06407=1023.717,98.128,392.926,167.800,48.819,159.062
C06408=1023.722,98.378,392.907,167.802,48.814,159.062
C06409=1023.728,98.627,392.889,167.804,48.809,159.061
C06410=1023.734,98.876,392.870,167.807,48.805,159.061
C06411=1023.740,99.126,392.852,167.810,48.800,159.060
C06412=1023.745,99.374,392.833,167.813,48.795,159.060
C06413=1023.751,99.624,392.815,167.815,48.791,159.059
C06414=1023.757,99.874,392.796,167.818,48.786,159.059
C06415=1023.762,100.122,392.777,167.821,48.781,159.058
C06416=1023.768,100.372,392.758,167.824,48.777,159.058
C06417=1023.774,100.621,392.740,167.826,48.773,159.057
C06418=1023.779,100.870,392.721,167.829,48.768,159.057
C06419=1023.786,101.119,392.703,167.832,48.763,159.056
C06420=1023.791,101.369,392.683,167.834,48.759,159.056
C06421=1023.797,101.618,392.664,167.837,48.754,159.055
C06422=1023.802,101.867,392.647,167.839,48.750,159.055
C06423=1023.808,102.117,392.627,167.843,48.745,159.054
C06424=1023.814,102.366,392.608,167.845,48.740,159.054
C06425=1023.820,102.615,392.590,167.848,48.736,159.053
C06426=1023.825,102.864,392.571,167.850,48.732,159.053
C06427=1023.831,103.114,392.552,167.854,48.727,159.052
C06428=1023.837,103.362,392.534,167.856,48.722,159.052
C06429=1023.842,103.612,392.515,167.858,48.718,159.051
C06430=1023.849,103.861,392.496,167.861,48.713,159.051
C06431=1023.854,104.110,392.477,167.864,48.708,159.050
C06432=1023.859,104.359,392.458,167.867,48.703,159.050
C06433=1023.866,104.608,392.439,167.869,48.699,159.049
C06434=1023.871,104.858,392.421,167.872,48.694,159.049
C06435=1023.877,105.108,392.401,167.875,48.689,159.048
C06436=1023.883,105.356,392.383,167.877,48.685,159.048
C06437=1023.888,105.606,392.364,167.880,48.680,159.047
C06438=1023.894,105.855,392.345,167.882,48.676,159.047
C06439=1023.901,106.104,392.326,167.886,48.671,159.046
C06440=1023.906,106.353,392.307,167.888,48.667,159.046
C06441=1023.911,106.602,392.288,167.891,48.662,159.045
C06442=1023.918,106.851,392.269,167.894,48.657,159.045
C06443=1023.923,107.101,392.250,167.897,48.653,159.044
C06444=1023.930,107.385,392.229,167.900,48.647,159.044
C06445=1023.937,107.669,392.207,167.903,48.642,159.043
C06446=1023.943,107.953,392.186,167.906,48.637,159.043
C06447=1023.950,108.237,392.164,167.908,48.632,159.042
C06448=1023.956,108.486,392.145,167.912,48.627,159.041
C06449=1023.961,108.735,392.126,167.914,48.622,159.041
C06450=1023.967,108.984,392.107,167.917,48.618,159.040
C06451=1023.973,109.233,392.088,167.920,48.613,159.040
C06452=1023.979,109.483,392.069,167.923,48.608,159.039
C06453=1023.985,109.732,392.050,167.925,48.604,159.039
C06454=1023.991,109.981,392.031,167.929,48.599,159.038
C06455=1023.996,110.230,392.012,167.931,48.594,159.038
C06456=1024.002,110.480,391.993,167.933,48.590,159.037
C06457=1024.007,110.729,391.973,167.936,48.585,159.037
C06458=1024.014,110.978,391.955,167.940,48.581,159.036
C06459=1024.019,111.228,391.936,167.942,48.576,159.036
C06460=1024.025,111.477,391.916,167.944,48.572,159.035
C06461=1024.030,111.726,391.897,167.948,48.567,159.035
C06462=1024.036,111.975,391.878,167.950,48.562,159.034
C06463=1024.043,112.224,391.859,167.953,48.558,159.034
C06464=1024.048,112.473,391.840,167.956,48.553,159.033
C06465=1024.054,112.723,391.820,167.959,48.548,159.033
C06466=1024.060,112.972,391.801,167.961,48.544,159.032
C06467=1024.065,113.222,391.781,167.964,48.540,159.032
C06468=1024.070,113.470,391.762,167.966,48.535,159.031
C06469=1024.076,113.719,391.742,167.970,48.530,159.031
C06470=1024.081,113.969,391.723,167.972,48.526,159.030
C06471=1024.087,114.218,391.703,167.975,48.522,159.030
C06472=1024.093,114.467,391.684,167.977,48.517,159.029
C06473=1024.099,114.716,391.665,167.981,48.513,159.029
C06474=1024.105,114.966,391.646,167.983,48.508,159.028
C06475=1024.110,115.214,391.626,167.986,48.503,159.028
C06476=1024.115,115.464,391.606,167.988,48.500,159.028
C06477=1024.121,115.713,391.587,167.992,48.495,159.027
C06478=1024.127,115.962,391.567,167.994,48.490,159.027
C06479=1024.132,116.211,391.548,167.997,48.486,159.026
C06480=1024.138,116.460,391.528,167.999,48.481,159.025
C06481=1024.144,116.710,391.508,168.003,48.477,159.025
C06482=1024.150,116.959,391.489,168.005,48.472,159.025
C06483=1024.155,117.207,391.470,168.008,48.468,159.024
C06484=1024.160,117.457,391.450,168.011,48.463,159.024
C06485=1024.166,117.706,391.431,168.014,48.458,159.023
C06486=1024.172,117.955,391.411,168.017,48.454,159.023
C06487=1024.177,118.205,391.391,168.019,48.450,159.022
C06488=1024.183,118.453,391.371,168.022,48.445,159.022
C06489=1024.189,118.703,391.352,168.025,48.441,159.021
C06490=1024.195,118.952,391.333,168.027,48.436,159.021
C06491=1024.201,119.201,391.313,168.031,48.431,159.020
C06492=1024.206,119.451,391.293,168.034,48.427,159.020
C06493=1024.212,119.700,391.273,168.036,48.423,159.019
C06494=1024.217,119.949,391.254,168.038,48.418,159.019
C06495=1024.223,120.198,391.234,168.042,48.413,159.018
C06496=1024.229,120.447,391.215,168.044,48.409,159.018
C06497=1024.235,120.696,391.195,168.047,48.404,159.017
C06498=1024.241,120.946,391.175,168.050,48.399,159.017
C06499=1024.246,121.195,391.155,168.053,48.395,159.016
C06500=1024.252,121.444,391.136,168.056,48.391,159.016
C06501=1024.258,121.693,391.116,168.059,48.386,159.015
C06502=1024.263,121.942,391.096,168.061,48.382,159.015
C06503=1024.269,122.191,391.077,168.064,48.377,159.014
C06504=1024.275,122.441,391.057,168.067,48.372,159.014
C06505=1024.281,122.689,391.037,168.070,48.368,159.013
C06506=1024.286,122.939,391.017,168.072,48.363,159.013
C06507=1024.292,123.188,390.998,168.076,48.359,159.012
C06508=1024.298,123.472,390.975,168.079,48.353,159.012
C06509=1024.305,123.755,390.953,168.082,48.348,159.011
C06510=1024.312,124.039,390.931,168.086,48.343,159.011
C06511=1024.319,124.323,390.908,168.089,48.338,159.010
C06512=1024.324,124.573,390.889,168.091,48.333,159.010
C06513=1024.330,124.822,390.868,168.094,48.329,159.009
C06514=1024.336,125.071,390.848,168.098,48.324,159.009
C06515=1024.341,125.320,390.829,168.100,48.320,159.008
C06516=1024.347,125.569,390.809,168.103,48.315,159.008
C06517=1024.353,125.818,390.790,168.106,48.310,159.007
C06518=1024.359,126.067,390.770,168.109,48.306,159.007
C06519=1024.364,126.316,390.749,168.112,48.301,159.006
C06520=1024.370,126.566,390.730,168.114,48.297,159.006
C06521=1024.376,126.815,390.710,168.117,48.292,159.005
C06522=1024.382,127.063,390.690,168.120,48.287,159.005
C06523=1024.388,127.313,390.671,168.123,48.283,159.004
C06524=1024.394,127.562,390.650,168.126,48.279,159.004
C06525=1024.399,127.811,390.630,168.129,48.274,159.003
C06526=1024.405,128.061,390.611,168.132,48.269,159.003
C06527=1024.411,128.310,390.591,168.135,48.265,159.002
C06528=1024.417,128.558,390.571,168.137,48.260,159.002
C06529=1024.423,128.808,390.551,168.140,48.256,159.001
C06530=1024.429,129.057,390.532,168.143,48.251,159.001
C06531=1024.434,129.306,390.511,168.146,48.246,159.000
C06532=1024.441,129.555,390.491,168.149,48.241,159.000
C06533=1024.446,129.805,390.471,168.152,48.237,158.999
C06534=1024.452,130.054,390.451,168.155,48.232,158.999
C06535=1024.458,130.302,390.431,168.158,48.228,158.998
C06536=1024.464,130.552,390.411,168.161,48.224,158.998
C06537=1024.470,130.800,390.391,168.164,48.219,158.997
C06538=1024.475,131.050,390.371,168.167,48.214,158.997
C06539=1024.481,131.299,390.351,168.169,48.210,158.996
C06540=1024.486,131.549,390.330,168.173,48.206,158.996
C06541=1024.492,131.798,390.310,168.175,48.201,158.995
C06542=1024.498,132.047,390.290,168.178,48.197,158.995
C06543=1024.504,132.295,390.270,168.181,48.192,158.994
C06544=1024.509,132.545,390.249,168.184,48.188,158.994
C06545=1024.515,132.793,390.229,168.187,48.183,158.993
C06546=1024.520,133.043,390.209,168.190,48.179,158.993
C06547=1024.527,133.292,390.188,168.192,48.174,158.992
C06548=1024.532,133.541,390.168,168.196,48.169,158.992
C06549=1024.538,133.790,390.148,168.199,48.166,158.992
C06550=1024.543,134.039,390.127,168.201,48.161,158.991
C06551=1024.549,134.288,390.107,168.205,48.156,158.991
C06552=1024.555,134.538,390.086,168.207,48.152,158.990
C06553=1024.561,134.787,390.066,168.211,48.148,158.990
C06554=1024.566,135.036,390.046,168.213,48.143,158.989
C06555=1024.572,135.284,390.026,168.216,48.139,158.989
C06556=1024.578,135.534,390.005,168.219,48.134,158.988
C06557=1024.584,135.783,389.985,168.222,48.129,158.988
C06558=1024.589,136.032,389.965,168.226,48.125,158.987
C06559=1024.595,136.281,389.944,168.228,48.121,158.987
C06560=1024.601,136.530,389.924,168.231,48.116,158.986
C06561=1024.606,136.779,389.903,168.234,48.111,158.986
C06562=1024.613,137.029,389.883,168.237,48.108,158.985
C06563=1024.618,137.278,389.863,168.240,48.103,158.985
C06564=1024.623,137.527,389.842,168.243,48.098,158.984
C06565=1024.629,137.775,389.821,168.245,48.094,158.984
C06566=1024.635,138.025,389.800,168.249,48.089,158.983
C06567=1024.641,138.274,389.780,168.252,48.085,158.983
C06568=1024.646,138.523,389.760,168.255,48.080,158.982
C06569=1024.652,138.772,389.739,168.258,48.076,158.982
C06570=1024.658,139.022,389.718,168.260,48.072,158.982
C06571=1024.664,139.270,389.698,168.264,48.067,158.981
C06572=1024.670,139.554,389.675,168.267,48.062,158.981
C06573=1024.676,139.838,389.651,168.271,48.057,158.980
C06574=1024.683,140.122,389.627,168.274,48.052,158.980
C06575=1024.689,140.406,389.603,168.278,48.047,158.979
C06576=1024.695,140.655,389.583,168.280,48.043,158.979
C06577=1024.701,140.904,389.563,168.284,48.038,158.978
C06578=1024.707,141.153,389.541,168.286,48.034,158.978
C06579=1024.712,141.402,389.521,168.290,48.029,158.977
C06580=1024.717,141.651,389.500,168.292,48.025,158.977
C06581=1024.724,141.901,389.480,168.295,48.020,158.976
C06582=1024.729,142.149,389.458,168.299,48.016,158.976
C06583=1024.735,142.398,389.438,168.301,48.012,158.975
C06584=1024.740,142.647,389.417,168.305,48.007,158.975
C06585=1024.746,142.896,389.396,168.307,48.003,158.974
C06586=1024.752,143.145,389.376,168.311,47.998,158.974
C06587=1024.757,143.394,389.355,168.313,47.994,158.973
C06588=1024.763,143.644,389.333,168.316,47.990,158.973
C06589=1024.769,143.893,389.313,168.320,47.985,158.973
C06590=1024.775,144.141,389.292,168.322,47.981,158.972
C06591=1024.781,144.391,389.271,168.326,47.976,158.972
C06592=1024.786,144.640,389.251,168.328,47.972,158.971
C06593=1024.792,144.889,389.229,168.332,47.968,158.971
C06594=1024.798,145.138,389.209,168.334,47.963,158.970
C06595=1024.804,145.386,389.188,168.338,47.959,158.970
C06596=1024.810,145.636,389.167,168.341,47.954,158.969
C06597=1024.815,145.885,389.146,168.344,47.950,158.969
C06598=1024.820,146.134,389.125,168.347,47.945,158.968
C06599=1024.826,146.384,389.104,168.351,47.941,158.968
C06600=1024.832,146.632,389.083,168.353,47.937,158.967
C06601=1024.838,146.882,389.062,168.356,47.933,158.967
C06602=1024.843,147.131,389.041,168.359,47.928,158.967
C06603=1024.849,147.379,389.020,168.362,47.924,158.966
C06604=1024.855,147.629,388.999,168.366,47.919,158.966
C06605=1024.860,147.877,388.977,168.368,47.915,158.965
C06606=1024.866,148.127,388.956,168.372,47.910,158.965
C06607=1024.872,148.376,388.935,168.375,47.906,158.964
C06608=1024.877,148.625,388.915,168.378,47.902,158.964
C06609=1024.883,148.874,388.893,168.381,47.898,158.963
C06610=1024.889,149.123,388.872,168.384,47.893,158.963
C06611=1024.895,149.372,388.851,168.387,47.889,158.962
C06612=1024.900,149.621,388.829,168.390,47.885,158.962
C06613=1024.906,149.869,388.808,168.393,47.880,158.962
C06614=1024.912,150.119,388.787,168.396,47.876,158.961
C06615=1024.917,150.368,388.766,168.400,47.871,158.961
C06616=1024.923,150.617,388.744,168.402,47.867,158.960
C06617=1024.929,150.866,388.724,168.406,47.863,158.960
C06618=1024.935,151.115,388.702,168.408,47.858,158.959
C06619=1024.940,151.364,388.681,168.412,47.854,158.959
C06620=1024.946,151.614,388.660,168.415,47.850,158.958
C06621=1024.952,151.862,388.639,168.418,47.845,158.958
C06622=1024.957,152.111,388.617,168.421,47.841,158.958
C06623=1024.963,152.360,388.596,168.425,47.837,158.957
C06624=1024.969,152.609,388.575,168.427,47.833,158.957
C06625=1024.975,152.858,388.554,168.431,47.828,158.956
C06626=1024.980,153.107,388.532,168.433,47.824,158.956
C06627=1024.986,153.356,388.510,168.437,47.819,158.955
C06628=1024.991,153.605,388.490,168.440,47.815,158.955
C06629=1024.997,153.854,388.468,168.444,47.811,158.955
C06630=1025.003,154.103,388.447,168.446,47.806,158.954
C06631=1025.009,154.352,388.425,168.450,47.802,158.954
C06632=1025.014,154.601,388.403,168.452,47.798,158.953
C06633=1025.020,154.850,388.382,168.456,47.794,158.953
C06634=1025.025,155.099,388.361,168.459,47.789,158.952
C06635=1025.031,155.348,388.339,168.463,47.785,158.952
C06636=1025.038,155.632,388.314,168.466,47.780,158.951
C06637=1025.044,155.915,388.290,168.469,47.775,158.951
C06638=1025.051,156.199,388.266,168.473,47.770,158.950
C06639=1025.058,156.482,388.241,168.476,47.766,158.950
C06640=1025.063,156.731,388.219,168.480,47.761,158.950
C06641=1025.069,156.980,388.197,168.484,47.757,158.949
C06642=1025.074,157.229,388.176,168.486,47.752,158.949
C06643=1025.081,157.478,388.155,168.490,47.748,158.948
C06644=1025.085,157.727,388.133,168.493,47.744,158.948
C06645=1025.091,157.976,388.111,168.496,47.740,158.947
C06646=1025.097,158.225,388.090,168.499,47.735,158.947
C06647=1025.103,158.474,388.068,168.503,47.731,158.947
C06648=1025.109,158.724,388.047,168.505,47.727,158.946
C06649=1025.114,158.973,388.025,168.509,47.722,158.946
C06650=1025.120,159.221,388.003,168.512,47.718,158.945
C06651=1025.125,159.470,387.981,168.515,47.714,158.945
C06652=1025.131,159.719,387.960,168.518,47.710,158.944
C06653=1025.137,159.969,387.937,168.522,47.706,158.944
C06654=1025.142,160.217,387.915,168.525,47.702,158.944
C06655=1025.148,160.467,387.894,168.528,47.697,158.943
C06656=1025.153,160.715,387.871,168.531,47.693,158.943
C06657=1025.158,160.964,387.849,168.535,47.689,158.943
C06658=1025.164,161.213,387.828,168.538,47.686,158.942
C06659=1025.169,161.462,387.805,168.541,47.681,158.942
C06660=1025.175,161.711,387.783,168.544,47.677,158.941
C06661=1025.181,161.960,387.761,168.548,47.673,158.941
C06662=1025.186,162.209,387.739,168.550,47.669,158.940
C06663=1025.191,162.458,387.716,168.554,47.664,158.940
C06664=1025.197,162.707,387.695,168.557,47.661,158.940
C06665=1025.203,162.956,387.673,168.561,47.656,158.939
C06666=1025.208,163.205,387.651,168.563,47.652,158.939
C06667=1025.214,163.454,387.628,168.567,47.648,158.939
C06668=1025.219,163.702,387.607,168.570,47.644,158.938
C06669=1025.224,163.952,387.584,168.574,47.640,158.938
C06670=1025.231,164.201,387.562,168.576,47.636,158.937
C06671=1025.236,164.449,387.540,168.580,47.632,158.937
C06672=1025.241,164.699,387.518,168.583,47.627,158.936
C06673=1025.247,164.947,387.496,168.587,47.623,158.936
C06674=1025.252,165.196,387.474,168.590,47.619,158.936
C06675=1025.258,165.445,387.451,168.593,47.615,158.935
C06676=1025.263,165.695,387.428,168.597,47.611,158.935
C06677=1025.269,165.943,387.407,168.600,47.607,158.935
C06678=1025.275,166.192,387.384,168.603,47.602,158.934
C06679=1025.280,166.442,387.362,168.606,47.599,158.934
C06680=1025.286,166.689,387.340,168.610,47.594,158.933
C06681=1025.291,166.939,387.318,168.612,47.590,158.933
C06682=1025.297,167.188,387.295,168.616,47.586,158.933
C06683=1025.303,167.437,387.273,168.620,47.582,158.932
C06684=1025.308,167.686,387.251,168.623,47.577,158.932
C06685=1025.314,167.935,387.228,168.626,47.573,158.931
C06686=1025.320,168.184,387.207,168.629,47.570,158.931
C06687=1025.326,168.433,387.184,168.633,47.566,158.931
C06688=1025.331,168.682,387.162,168.637,47.561,158.930
C06689=1025.336,168.931,387.139,168.640,47.557,158.930
C06690=1025.343,169.180,387.117,168.643,47.553,158.930
C06691=1025.348,169.429,387.094,168.646,47.549,158.929
C06692=1025.353,169.677,387.072,168.650,47.545,158.929
C06693=1025.360,169.926,387.050,168.654,47.541,158.928
C06694=1025.365,170.175,387.027,168.656,47.536,158.928
C06695=1025.371,170.425,387.005,168.660,47.532,158.927
C06696=1025.376,170.673,386.982,168.664,47.528,158.927
C06697=1025.382,170.922,386.961,168.667,47.524,158.927
C06698=1025.388,171.171,386.938,168.670,47.520,158.926
C06699=1025.393,171.420,386.915,168.674,47.516,158.926
C06700=1025.400,171.703,386.890,168.678,47.511,158.926
C06701=1025.406,171.986,386.865,168.681,47.506,158.925
C06702=1025.413,172.269,386.839,168.685,47.502,158.925
C06703=1025.419,172.552,386.813,168.689,47.497,158.924
C06704=1025.426,172.801,386.791,168.692,47.493,158.924
C06705=1025.431,173.051,386.769,168.696,47.489,158.923
C06706=1025.436,173.299,386.746,168.700,47.484,158.923
C06707=1025.442,173.548,386.723,168.702,47.480,158.923
C06708=1025.448,173.797,386.701,168.706,47.476,158.922
C06709=1025.454,174.046,386.679,168.710,47.472,158.922
C06710=1025.460,174.295,386.656,168.714,47.468,158.921
C06711=1025.466,174.544,386.634,168.716,47.464,158.921
C06712=1025.472,174.793,386.611,168.720,47.460,158.921
C06713=1025.477,175.042,386.588,168.724,47.455,158.920
C06714=1025.483,175.291,386.565,168.727,47.451,158.920
C06715=1025.489,175.539,386.544,168.731,47.447,158.920
C06716=1025.494,175.788,386.521,168.734,47.443,158.919
C06717=1025.500,176.037,386.498,168.738,47.439,158.919
C06718=1025.506,176.286,386.475,168.741,47.435,158.918
C06719=1025.512,176.535,386.453,168.745,47.431,158.918
C06720=1025.518,176.784,386.430,168.748,47.426,158.918
C06721=1025.523,177.033,386.407,168.751,47.422,158.917
C06722=1025.529,177.282,386.385,168.755,47.418,158.917
C06723=1025.536,177.530,386.362,168.758,47.414,158.916
C06724=1025.541,177.780,386.340,168.762,47.410,158.916
C06725=1025.547,178.029,386.317,168.765,47.406,158.916
C06726=1025.553,178.277,386.295,168.769,47.402,158.915
C06727=1025.559,178.526,386.272,168.773,47.397,158.915
C06728=1025.565,178.775,386.249,168.776,47.393,158.915
C06729=1025.570,179.024,386.226,168.780,47.389,158.914
C06730=1025.577,179.272,386.203,168.783,47.385,158.914
C06731=1025.582,179.522,386.181,168.787,47.381,158.913
C06732=1025.588,179.771,386.158,168.791,47.377,158.913
C06733=1025.594,180.020,386.135,168.794,47.373,158.913
C06734=1025.600,180.268,386.113,168.798,47.368,158.912
C06735=1025.606,180.517,386.090,168.801,47.364,158.912
C06736=1025.612,180.766,386.067,168.805,47.360,158.912
C06737=1025.617,181.015,386.044,168.809,47.356,158.911
C06738=1025.624,181.264,386.022,168.812,47.352,158.911
C06739=1025.630,181.513,385.999,168.816,47.348,158.910
C06740=1025.635,181.761,385.976,168.819,47.344,158.910
C06741=1025.641,182.010,385.953,168.823,47.340,158.910
C06742=1025.648,182.260,385.930,168.826,47.335,158.909
C06743=1025.654,182.509,385.907,168.830,47.331,158.909
C06744=1025.660,182.757,385.884,168.834,47.327,158.909
C06745=1025.665,183.007,385.861,168.837,47.323,158.908
C06746=1025.670,183.256,385.838,168.841,47.319,158.908
C06747=1025.676,183.504,385.814,168.845,47.315,158.908
C06748=1025.681,183.753,385.791,168.847,47.312,158.907
C06749=1025.687,184.002,385.768,168.851,47.308,158.907
C06750=1025.692,184.250,385.743,168.855,47.304,158.907
C06751=1025.698,184.499,385.721,168.859,47.300,158.906
C06752=1025.703,184.749,385.697,168.862,47.297,158.906
C06753=1025.709,184.997,385.674,168.866,47.293,158.906
C06754=1025.715,185.246,385.650,168.870,47.289,158.905
C06755=1025.720,185.495,385.627,168.873,47.285,158.905
C06756=1025.726,185.743,385.603,168.877,47.281,158.905
C06757=1025.732,185.992,385.580,168.881,47.277,158.904
C06758=1025.737,186.242,385.556,168.884,47.273,158.904
C06759=1025.743,186.490,385.533,168.887,47.269,158.904
C06760=1025.749,186.739,385.510,168.891,47.265,158.903
C06761=1025.754,186.988,385.486,168.895,47.261,158.903
C06762=1025.760,187.237,385.463,168.899,47.257,158.903
C06763=1025.765,187.486,385.439,168.903,47.254,158.903
C06764=1025.772,187.768,385.412,168.907,47.249,158.902
C06765=1025.779,188.051,385.385,168.910,47.245,158.902
C06766=1025.784,188.333,385.359,168.915,47.240,158.901
C06767=1025.791,188.616,385.332,168.919,47.236,158.901
C06768=1025.796,188.865,385.308,168.923,47.232,158.901
C06769=1025.803,189.114,385.285,168.927,47.228,158.900
C06770=1025.809,189.363,385.261,168.931,47.224,158.900
C06771=1025.814,189.612,385.238,168.934,47.220,158.900
C06772=1025.820,189.860,385.214,168.937,47.217,158.899
C06773=1025.825,190.109,385.191,168.941,47.213,158.899
C06774=1025.831,190.358,385.167,168.945,47.209,158.899
C06775=1025.837,190.607,385.143,168.949,47.205,158.899
C06776=1025.842,190.856,385.119,168.953,47.201,158.898
C06777=1025.848,191.104,385.096,168.956,47.198,158.898
C06778=1025.854,191.353,385.073,168.960,47.194,158.897
C06779=1025.860,191.602,385.048,168.964,47.190,158.897
C06780=1025.866,191.851,385.025,168.968,47.186,158.897
C06781=1025.871,192.100,385.001,168.971,47.182,158.897
C06782=1025.877,192.348,384.977,168.975,47.178,158.896
C06783=1025.883,192.597,384.954,168.979,47.174,158.896
C06784=1025.889,192.846,384.930,168.982,47.171,158.896
C06785=1025.895,193.094,384.906,168.986,47.167,158.895
C06786=1025.900,193.344,384.882,168.990,47.163,158.895
C06787=1025.906,193.593,384.858,168.994,47.159,158.895
C06788=1025.912,193.841,384.834,168.998,47.155,158.894
C06789=1025.917,194.090,384.811,169.002,47.151,158.894
C06790=1025.924,194.338,384.788,169.006,47.147,158.894
C06791=1025.929,194.588,384.763,169.010,47.143,158.894
C06792=1025.935,194.836,384.739,169.014,47.140,158.893
C06793=1025.940,195.085,384.716,169.018,47.136,158.893
C06794=1025.947,195.334,384.692,169.020,47.132,158.892
C06795=1025.953,195.582,384.668,169.024,47.128,158.892
C06796=1025.958,195.831,384.644,169.028,47.125,158.892
C06797=1025.965,196.081,384.620,169.032,47.121,158.892
C06798=1025.970,196.329,384.596,169.036,47.117,158.891
C06799=1025.976,196.577,384.573,169.040,47.113,158.891
C06800=1025.982,196.827,384.548,169.044,47.109,158.891
C06801=1025.988,197.075,384.524,169.048,47.105,158.890
C06802=1025.994,197.325,384.501,169.052,47.101,158.890
C06803=1026.000,197.573,384.477,169.056,47.097,158.890
C06804=1026.006,197.808,384.454,169.060,47.093,158.890
C06805=1026.011,198.043,384.431,169.063,47.090,158.889
C06806=1026.017,198.278,384.409,169.067,47.086,158.889
C06807=1026.022,198.513,384.386,169.071,47.082,158.889
C06808=1026.028,198.749,384.363,169.074,47.079,158.888
C06809=1026.034,198.983,384.341,169.078,47.075,158.888
C06810=1026.039,199.219,384.318,169.082,47.072,158.888
C06811=1026.045,199.453,384.295,169.086,47.068,158.888
C06812=1026.050,199.702,384.271,169.090,47.064,158.887
C06813=1026.057,199.951,384.247,169.094,47.060,158.887
C06814=1026.062,200.200,384.223,169.098,47.057,158.887
C06815=1026.068,200.449,384.198,169.101,47.053,158.886
C06816=1026.074,200.697,384.174,169.105,47.050,158.886
C06817=1026.080,200.946,384.150,169.109,47.046,158.886
C06818=1026.085,201.195,384.126,169.113,47.042,158.886
C06819=1026.091,201.444,384.101,169.117,47.039,158.885
C06820=1026.097,201.693,384.077,169.121,47.035,158.885
C06821=1026.103,201.941,384.053,169.125,47.031,158.885
C06822=1026.109,202.190,384.028,169.129,47.027,158.885
C06823=1026.114,202.438,384.003,169.133,47.024,158.884
C06824=1026.120,202.688,383.979,169.137,47.020,158.884
C06825=1026.125,202.936,383.955,169.141,47.016,158.884
C06826=1026.132,203.185,383.930,169.145,47.013,158.884
C06827=1026.138,203.433,383.906,169.149,47.009,158.883
C06828=1026.164,204.581,383.792,169.542,47.110,158.954
C06829=1026.175,204.976,383.752,169.547,47.105,158.954
C06830=1026.186,205.372,383.710,169.551,47.100,158.953
C06831=1026.196,205.769,383.669,169.556,47.096,158.953
C06832=1026.207,206.165,383.627,169.561,47.091,158.952
C06833=1026.213,206.413,383.601,169.564,47.089,158.952
C06834=1026.220,206.663,383.576,169.567,47.086,158.952
C06835=1026.227,206.911,383.549,169.570,47.083,158.952
C06836=1026.232,207.159,383.523,169.573,47.080,158.952
C06837=1026.240,207.408,383.496,169.576,47.078,158.951
C06838=1026.246,207.657,383.471,169.579,47.075,158.951
C06839=1026.253,207.905,383.445,169.582,47.072,158.951
C06840=1026.259,208.153,383.419,169.585,47.069,158.951
C06841=1026.266,208.402,383.392,169.588,47.066,158.951
C06842=1026.272,208.651,383.366,169.591,47.063,158.950
C06843=1026.278,208.899,383.340,169.594,47.060,158.950
C06844=1026.286,209.148,383.314,169.598,47.058,158.950
C06845=1026.292,209.396,383.288,169.600,47.055,158.950
C06846=1026.299,209.645,383.261,169.603,47.052,158.949
C06847=1026.305,209.894,383.235,169.607,47.050,158.949
C06848=1026.312,210.142,383.209,169.610,47.047,158.949
C06849=1026.318,210.390,383.183,169.613,47.044,158.949
C06850=1026.325,210.639,383.156,169.615,47.042,158.949
C06851=1026.331,210.888,383.130,169.618,47.039,158.948
C06852=1026.338,211.136,383.104,169.622,47.036,158.948
C06853=1026.345,211.384,383.077,169.625,47.033,158.948
C06854=1026.351,211.633,383.051,169.628,47.030,158.948
C06855=1026.358,211.881,383.024,169.631,47.028,158.948
C06856=1026.363,212.130,382.998,169.634,47.025,158.948
C06857=1026.371,212.379,382.971,169.637,47.023,158.947
C06858=1026.377,212.627,382.945,169.640,47.020,158.947
C06859=1026.383,212.876,382.918,169.643,47.018,158.947
C06860=1026.390,213.124,382.892,169.646,47.015,158.947
C06861=1026.396,213.373,382.865,169.649,47.012,158.947
C06862=1026.403,213.621,382.839,169.653,47.009,158.946
C06863=1026.409,213.870,382.812,169.656,47.007,158.946
C06864=1026.416,214.118,382.786,169.658,47.004,158.946
C06865=1026.423,214.367,382.760,169.662,47.002,158.946
C06866=1026.429,214.615,382.733,169.665,46.999,158.946
C06867=1026.436,214.864,382.706,169.668,46.996,158.946
C06868=1026.442,215.112,382.680,169.671,46.993,158.945
C06869=1026.449,215.361,382.653,169.674,46.991,158.945
C06870=1026.456,215.610,382.627,169.677,46.988,158.945
C06871=1026.462,215.858,382.600,169.680,46.986,158.945
C06872=1026.469,216.107,382.574,169.683,46.983,158.945
C06873=1026.475,216.354,382.547,169.687,46.980,158.945
C06874=1026.482,216.603,382.520,169.690,46.977,158.944
C06875=1026.488,216.851,382.494,169.693,46.975,158.944
C06876=1026.495,217.100,382.467,169.696,46.972,158.944
C06877=1026.502,217.349,382.441,169.699,46.970,158.944
C06878=1026.508,217.597,382.414,169.702,46.967,158.944
C06879=1026.515,217.846,382.388,169.706,46.965,158.944
C06880=1026.521,218.094,382.360,169.708,46.962,158.943
C06881=1026.528,218.343,382.334,169.711,46.959,158.943
C06882=1026.535,218.591,382.307,169.715,46.957,158.943
C06883=1026.541,218.840,382.281,169.718,46.954,158.943
C06884=1026.548,219.088,382.254,169.721,46.952,158.943
C06885=1026.558,219.488,382.210,169.726,46.947,158.943
C06886=1026.568,219.888,382.167,169.731,46.943,158.942
C06887=1026.579,220.287,382.124,169.736,46.940,158.942
C06888=1026.589,220.687,382.080,169.741,46.936,158.942
C06889=1026.596,220.936,382.054,169.745,46.933,158.942
C06890=1026.603,221.184,382.026,169.748,46.931,158.942
C06891=1026.608,221.433,382.000,169.751,46.928,158.941
C06892=1026.616,221.681,381.972,169.754,46.926,158.941
C06893=1026.622,221.930,381.945,169.757,46.923,158.941
C06894=1026.628,222.178,381.919,169.761,46.921,158.941
C06895=1026.635,222.427,381.891,169.764,46.918,158.941
C06896=1026.642,222.675,381.865,169.767,46.916,158.941
C06897=1026.648,222.923,381.837,169.770,46.914,158.941
C06898=1026.654,223.172,381.810,169.773,46.911,158.941
C06899=1026.662,223.420,381.783,169.776,46.908,158.940
C06900=1026.667,223.669,381.756,169.780,46.906,158.940
C06901=1026.674,223.917,381.729,169.783,46.903,158.940
C06902=1026.680,224.166,381.702,169.787,46.901,158.940
C06903=1026.688,224.414,381.675,169.789,46.899,158.940
C06904=1026.694,224.663,381.648,169.792,46.896,158.940
C06905=1026.700,224.911,381.620,169.796,46.894,158.940
C06906=1026.707,225.160,381.594,169.799,46.891,158.940
C06907=1026.713,225.408,381.566,169.803,46.889,158.939
C06908=1026.720,225.657,381.539,169.806,46.887,158.939
C06909=1026.727,225.905,381.512,169.808,46.884,158.939
C06910=1026.734,226.154,381.485,169.812,46.881,158.939
C06911=1026.740,226.402,381.458,169.815,46.879,158.939
C06912=1026.746,226.650,381.430,169.819,46.877,158.939
C06913=1026.754,226.899,381.404,169.822,46.874,158.939
C06914=1026.760,227.147,381.376,169.825,46.872,158.939
C06915=1026.766,227.395,381.349,169.828,46.870,158.939
C06916=1026.773,227.644,381.322,169.831,46.868,158.938
C06917=1026.779,227.892,381.294,169.835,46.865,158.938
C06918=1026.786,228.141,381.266,169.838,46.862,158.938
C06919=1026.792,228.389,381.239,169.841,46.860,158.938
C06920=1026.798,228.638,381.212,169.844,46.858,158.938
C06921=1026.805,228.886,381.184,169.847,46.855,158.938
C06922=1026.812,229.135,381.156,169.851,46.853,158.938
C06923=1026.818,229.384,381.129,169.854,46.851,158.938
C06924=1026.824,229.631,381.102,169.858,46.848,158.938
C06925=1026.831,229.880,381.074,169.861,46.846,158.937
C06926=1026.838,230.128,381.046,169.864,46.844,158.937
C06927=1026.845,230.376,381.019,169.867,46.842,158.937
C06928=1026.852,230.625,380.992,169.870,46.839,158.937
C06929=1026.858,230.873,380.965,169.874,46.838,158.937
C06930=1026.863,231.122,380.937,169.878,46.835,158.937
C06931=1026.870,231.370,380.909,169.881,46.833,158.937
C06932=1026.877,231.619,380.881,169.884,46.831,158.937
C06933=1026.884,231.867,380.853,169.887,46.828,158.937
C06934=1026.890,232.116,380.826,169.890,46.826,158.937
C06935=1026.896,232.363,380.798,169.894,46.824,158.937
C06936=1026.903,232.612,380.771,169.897,46.821,158.937
C06937=1026.910,232.860,380.743,169.900,46.819,158.936
C06938=1026.916,233.109,380.715,169.904,46.818,158.937
C06939=1026.922,233.358,380.687,169.907,46.815,158.936
C06940=1026.929,233.606,380.659,169.910,46.813,158.936
C06941=1026.939,233.998,380.616,169.916,46.809,158.936
C06942=1026.950,234.390,380.572,169.921,46.806,158.936
C06943=1026.960,234.782,380.528,169.926,46.802,158.936
C06944=1026.970,235.174,380.484,169.931,46.799,158.936
C06945=1026.977,235.423,380.456,169.935,46.796,158.936
C06946=1026.983,235.671,380.428,169.938,46.795,158.936
C06947=1026.990,235.919,380.401,169.942,46.792,158.936
C06948=1026.997,236.168,380.373,169.945,46.790,158.936
C06949=1027.003,236.416,380.346,169.948,46.788,158.936
C06950=1027.010,236.663,380.317,169.951,46.786,158.936
C06951=1027.016,236.912,380.289,169.955,46.784,158.936
C06952=1027.022,237.161,380.261,169.958,46.782,158.936
C06953=1027.029,237.409,380.233,169.962,46.779,158.935
C06954=1027.036,237.658,380.206,169.965,46.777,158.935
C06955=1027.042,237.906,380.178,169.969,46.775,158.935
C06956=1027.049,238.154,380.149,169.973,46.773,158.935
C06957=1027.055,238.403,380.121,169.975,46.771,158.935
C06958=1027.062,238.651,380.093,169.978,46.768,158.935
C06959=1027.069,238.899,380.066,169.982,46.767,158.935
C06960=1027.076,239.147,380.037,169.986,46.764,158.935
C06961=1027.082,239.396,380.009,169.989,46.762,158.935
C06962=1027.088,239.644,379.981,169.993,46.760,158.935
C06963=1027.095,239.893,379.953,169.996,46.758,158.935
C06964=1027.102,240.141,379.925,169.999,46.756,158.935
C06965=1027.108,240.389,379.897,170.003,46.754,158.935
C06966=1027.115,240.638,379.869,170.006,46.752,158.935
C06967=1027.121,240.886,379.840,170.010,46.750,158.935
C06968=1027.128,241.134,379.812,170.013,46.748,158.935
C06969=1027.134,241.383,379.783,170.017,46.746,158.935
C06970=1027.141,241.631,379.755,170.020,46.744,158.935
C06971=1027.147,241.879,379.726,170.023,46.742,158.935
C06972=1027.153,242.128,379.699,170.027,46.740,158.935
C06973=1027.160,242.375,379.670,170.030,46.738,158.935
C06974=1027.166,242.624,379.642,170.034,46.736,158.935
C06975=1027.173,242.873,379.614,170.037,46.734,158.935
C06976=1027.179,243.121,379.585,170.041,46.732,158.935
C06977=1027.186,243.369,379.557,170.044,46.730,158.935
C06978=1027.192,243.617,379.528,170.047,46.728,158.935
C06979=1027.199,243.865,379.500,170.051,46.726,158.935
C06980=1027.205,244.114,379.472,170.054,46.724,158.935
C06981=1027.212,244.362,379.443,170.058,46.722,158.935
C06982=1027.218,244.610,379.415,170.062,46.720,158.935
C06983=1027.224,244.859,379.386,170.065,46.718,158.935
C06984=1027.231,245.107,379.356,170.068,46.716,158.935
C06985=1027.238,245.356,379.329,170.072,46.715,158.935
C06986=1027.244,245.604,379.300,170.075,46.712,158.935
C06987=1027.250,245.852,379.270,170.079,46.711,158.935
C06988=1027.257,246.100,379.241,170.083,46.709,158.935
C06989=1027.263,246.349,379.214,170.086,46.707,158.935
C06990=1027.270,246.597,379.185,170.090,46.705,158.935
C06991=1027.276,246.845,379.156,170.092,46.704,158.935
C06992=1027.283,247.093,379.127,170.096,46.701,158.935
C06993=1027.289,247.342,379.099,170.100,46.700,158.935
C06994=1027.295,247.590,379.070,170.103,46.698,158.935
C06995=1027.302,247.839,379.040,170.107,46.696,158.935
C06996=1027.309,248.086,379.012,170.111,46.694,158.935
C06997=1027.318,248.472,378.967,170.116,46.691,158.935
C06998=1027.328,248.858,378.922,170.122,46.688,158.935
C06999=1027.338,249.244,378.877,170.127,46.685,158.935
C07000=1027.348,249.630,378.832,170.133,46.682,158.935
C07001=1027.355,249.878,378.804,170.136,46.681,158.935
C07002=1027.362,250.126,378.775,170.140,46.679,158.935
C07003=1027.368,250.375,378.746,170.143,46.677,158.935
C07004=1027.374,250.623,378.717,170.146,46.675,158.935
C07005=1027.381,250.871,378.689,170.150,46.674,158.935
C07006=1027.388,251.119,378.660,170.154,46.672,158.935
C07007=1027.394,251.368,378.630,170.157,46.670,158.935
C07008=1027.401,251.616,378.601,170.161,46.668,158.935
C07009=1027.408,251.864,378.573,170.165,46.666,158.936
C07010=1027.414,252.112,378.544,170.168,46.665,158.936
C07011=1027.421,252.361,378.514,170.172,46.663,158.936
C07012=1027.427,252.609,378.485,170.176,46.661,158.936
C07013=1027.433,252.857,378.456,170.178,46.659,158.936
C07014=1027.440,253.105,378.428,170.182,46.657,158.936
C07015=1027.447,253.354,378.399,170.186,46.656,158.936
C07016=1027.453,253.602,378.369,170.190,46.654,158.936
C07017=1027.460,253.850,378.340,170.193,46.652,158.936
C07018=1027.467,254.098,378.312,170.197,46.650,158.936
C07019=1027.473,254.347,378.283,170.201,46.648,158.936
C07020=1027.480,254.595,378.254,170.204,46.647,158.936
C07021=1027.486,254.843,378.225,170.208,46.645,158.936
C07022=1027.494,255.091,378.195,170.212,46.643,158.936
C07023=1027.500,255.339,378.166,170.216,46.642,158.936
C07024=1027.506,255.587,378.137,170.219,46.640,158.936
C07025=1027.513,255.836,378.107,170.223,46.638,158.936
C07026=1027.519,256.084,378.078,170.227,46.636,158.936
C07027=1027.526,256.332,378.050,170.230,46.634,158.936
C07028=1027.533,256.581,378.021,170.234,46.633,158.937
C07029=1027.540,256.828,377.991,170.238,46.631,158.937
C07030=1027.547,257.077,377.961,170.242,46.629,158.937
C07031=1027.554,257.325,377.933,170.244,46.628,158.937
C07032=1027.560,257.573,377.904,170.248,46.626,158.937
C07033=1027.567,257.822,377.875,170.252,46.624,158.937
C07034=1027.573,258.070,377.845,170.256,46.623,158.937
C07035=1027.580,258.318,377.815,170.259,46.621,158.937
C07036=1027.587,258.566,377.787,170.263,46.619,158.937
C07037=1027.593,258.814,377.758,170.267,46.617,158.937
C07038=1027.600,259.063,377.728,170.270,46.615,158.937
C07039=1027.607,259.311,377.699,170.274,46.614,158.937
C07040=1027.614,259.560,377.669,170.278,46.612,158.937
C07041=1027.621,259.807,377.640,170.282,46.610,158.937
C07042=1027.628,260.056,377.611,170.285,46.609,158.937
C07043=1027.634,260.304,377.582,170.289,46.607,158.938
C07044=1027.641,260.552,377.552,170.293,46.605,158.938
C07045=1027.648,260.800,377.523,170.297,46.604,158.938
C07046=1027.655,261.047,377.493,170.300,46.602,158.938
C07047=1027.661,261.296,377.463,170.304,46.601,158.938
C07048=1027.667,261.544,377.434,170.308,46.599,158.938
C07049=1027.674,261.793,377.404,170.312,46.597,158.938
C07050=1027.681,262.040,377.374,170.316,46.596,158.938
C07051=1027.688,262.289,377.345,170.319,46.594,158.938
C07052=1027.693,262.537,377.315,170.323,46.593,158.939
C07053=1027.704,262.921,377.269,170.329,46.590,158.939
C07054=1027.714,263.305,377.223,170.335,46.588,158.939
C07055=1027.725,263.690,377.177,170.340,46.586,158.939
C07056=1027.735,264.075,377.130,170.347,46.583,158.939
C07057=1027.741,264.323,377.101,170.351,46.582,158.939
C07058=1027.748,264.571,377.071,170.355,46.580,158.940
C07059=1027.755,264.819,377.041,170.359,46.579,158.940
C07060=1027.762,265.067,377.011,170.362,46.577,158.940
C07061=1027.767,265.315,376.981,170.366,46.576,158.940
C07062=1027.774,265.563,376.951,170.370,46.574,158.940
C07063=1027.781,265.811,376.921,170.374,46.573,158.940
C07064=1027.788,266.060,376.892,170.378,46.571,158.940
C07065=1027.794,266.308,376.862,170.382,46.569,158.940
C07066=1027.801,266.556,376.831,170.386,46.568,158.941
C07067=1027.808,266.804,376.801,170.388,46.567,158.941
C07068=1027.814,267.052,376.771,170.392,46.566,158.941
C07069=1027.821,267.300,376.741,170.396,46.564,158.941
C07070=1027.828,267.548,376.711,170.400,46.563,158.941
C07071=1027.834,267.797,376.681,170.404,46.562,158.941
C07072=1027.840,268.044,376.651,170.408,46.560,158.941
C07073=1027.847,268.292,376.621,170.412,46.559,158.942
C07074=1027.854,268.541,376.590,170.415,46.557,158.942
C07075=1027.860,268.788,376.561,170.419,46.556,158.942
C07076=1027.867,269.037,376.531,170.423,46.554,158.942
C07077=1027.873,269.284,376.500,170.427,46.553,158.942
C07078=1027.880,269.533,376.470,170.432,46.552,158.943
C07079=1027.888,269.781,376.440,170.436,46.550,158.943
C07080=1027.893,270.029,376.410,170.440,46.549,158.943
C07081=1027.901,270.277,376.380,170.444,46.547,158.943
C07082=1027.907,270.525,376.349,170.448,46.546,158.943
C07083=1027.914,270.773,376.319,170.451,46.544,158.943
C07084=1027.920,271.021,376.288,170.455,46.543,158.944
C07085=1027.927,271.269,376.258,170.459,46.542,158.944
C07086=1027.933,271.517,376.227,170.463,46.541,158.944
C07087=1027.940,271.765,376.197,170.467,46.540,158.944
C07088=1027.947,272.014,376.166,170.471,46.538,158.944
C07089=1027.953,272.261,376.137,170.475,46.537,158.944
C07090=1027.960,272.510,376.106,170.479,46.536,158.945
C07091=1027.967,272.757,376.075,170.483,46.534,158.945
C07092=1027.973,273.005,376.045,170.487,46.533,158.945
C07093=1027.980,273.254,376.014,170.491,46.531,158.945
C07094=1027.987,273.502,375.984,170.495,46.530,158.945
C07095=1027.993,273.749,375.953,170.499,46.529,158.946
C07096=1028.000,273.997,375.923,170.502,46.528,158.946
C07097=1028.006,274.246,375.892,170.506,46.527,158.946
C07098=1028.013,274.494,375.861,170.511,46.526,158.946
C07099=1028.020,274.741,375.831,170.514,46.524,158.946
C07100=1028.026,274.990,375.800,170.518,46.523,158.946
C07101=1028.033,275.238,375.770,170.522,46.522,158.947
C07102=1028.040,275.486,375.738,170.526,46.521,158.947
C07103=1028.046,275.734,375.708,170.530,46.519,158.947
C07104=1028.053,275.981,375.677,170.534,46.518,158.947
C07105=1028.060,276.230,375.647,170.538,46.517,158.948
C07106=1028.066,276.478,375.616,170.542,46.516,158.948
C07107=1028.074,276.726,375.585,170.547,46.514,158.948
C07108=1028.079,276.974,375.555,170.551,46.513,158.948
C07109=1028.090,277.363,375.506,170.557,46.512,158.949
C07110=1028.101,277.751,375.458,170.563,46.510,158.949
C07111=1028.111,278.141,375.409,170.570,46.508,158.949
C07112=1028.121,278.530,375.361,170.576,46.506,158.950
C07113=1028.128,278.778,375.329,170.580,46.505,158.950
C07114=1028.135,279.026,375.298,170.584,46.504,158.950
C07115=1028.142,279.274,375.268,170.588,46.503,158.950
C07116=1028.148,279.522,375.236,170.592,46.502,158.951
C07117=1028.155,279.769,375.205,170.596,46.501,158.951
C07118=1028.161,280.018,375.174,170.600,46.500,158.951
C07119=1028.168,280.266,375.143,170.605,46.498,158.951
C07120=1028.174,280.514,375.112,170.609,46.497,158.952
C07121=1028.181,280.762,375.081,170.613,46.496,158.952
C07122=1028.188,281.010,375.050,170.617,46.495,158.952
C07123=1028.195,281.258,375.019,170.621,46.494,158.952
C07124=1028.202,281.506,374.987,170.626,46.493,158.953
C07125=1028.208,281.753,374.957,170.630,46.492,158.953
C07126=1028.214,282.001,374.925,170.634,46.491,158.953
C07127=1028.221,282.249,374.894,170.638,46.490,158.953
C07128=1028.228,282.497,374.862,170.642,46.489,158.954
C07129=1028.234,282.745,374.831,170.647,46.488,158.954
C07130=1028.242,282.993,374.800,170.651,46.487,158.954
C07131=1028.248,283.241,374.769,170.655,46.486,158.954
C07132=1028.255,283.489,374.738,170.659,46.485,158.955
C07133=1028.262,283.737,374.707,170.663,46.484,158.955
C07134=1028.269,283.985,374.675,170.667,46.483,158.955
C07135=1028.275,284.233,374.644,170.671,46.482,158.955
C07136=1028.282,284.481,374.612,170.675,46.481,158.956
C07137=1028.289,284.728,374.581,170.680,46.479,158.956
C07138=1028.295,284.976,374.549,170.684,46.479,158.956
C07139=1028.302,285.224,374.518,170.688,46.478,158.957
C07140=1028.310,285.472,374.487,170.692,46.477,158.957
C07141=1028.316,285.720,374.456,170.697,46.476,158.957
C07142=1028.323,285.968,374.424,170.701,46.475,158.957
C07143=1028.330,286.216,374.393,170.705,46.474,158.958
C07144=1028.336,286.464,374.361,170.710,46.473,158.958
C07145=1028.343,286.712,374.329,170.714,46.472,158.958
C07146=1028.349,286.960,374.298,170.718,46.471,158.959
C07147=1028.356,287.208,374.267,170.722,46.470,158.959
C07148=1028.363,287.455,374.234,170.726,46.470,158.959
C07149=1028.370,287.703,374.203,170.730,46.468,158.960
C07150=1028.377,287.951,374.171,170.734,46.467,158.960
C07151=1028.384,288.199,374.140,170.740,46.467,158.960
C07152=1028.390,288.447,374.108,170.744,46.466,158.961
C07153=1028.397,288.695,374.076,170.748,46.465,158.961
C07154=1028.404,288.943,374.044,170.752,46.464,158.961
C07155=1028.410,289.191,374.013,170.756,46.463,158.961
C07156=1028.417,289.438,373.981,170.760,46.462,158.962
C07157=1028.424,289.686,373.949,170.766,46.462,158.962
C07158=1028.431,289.934,373.918,170.770,46.461,158.962
C07159=1028.437,290.183,373.885,170.774,46.460,158.963
C07160=1028.444,290.430,373.853,170.778,46.459,158.963
C07161=1028.451,290.678,373.822,170.782,46.458,158.963
C07162=1028.458,290.925,373.790,170.787,46.457,158.964
C07163=1028.465,291.173,373.758,170.791,46.456,158.964
C07164=1028.471,291.421,373.726,170.796,46.456,158.964
C07165=1028.483,291.823,373.674,170.803,46.454,158.965
C07166=1028.494,292.223,373.622,170.810,46.453,158.966
C07167=1028.504,292.625,373.571,170.817,46.452,158.966
C07168=1028.515,293.026,373.519,170.824,46.451,158.967
C07169=1028.522,293.274,373.486,170.828,46.450,158.967
C07170=1028.529,293.522,373.454,170.833,46.449,158.967
C07171=1028.536,293.769,373.422,170.838,46.449,158.968
C07172=1028.542,294.018,373.390,170.842,46.448,158.968
C07173=1028.549,294.265,373.358,170.846,46.447,158.968
C07174=1028.555,294.513,373.325,170.850,46.446,158.969
C07175=1028.563,294.760,373.293,170.855,46.446,158.969
C07176=1028.569,295.009,373.261,170.860,46.445,158.970
C07177=1028.575,295.256,373.228,170.864,46.445,158.970
C07178=1028.582,295.504,373.196,170.868,46.444,158.970
C07179=1028.589,295.752,373.163,170.872,46.443,158.971
C07180=1028.596,295.999,373.130,170.877,46.443,158.971
C07181=1028.603,296.247,373.098,170.882,46.442,158.972
C07182=1028.609,296.495,373.066,170.886,46.442,158.972
C07183=1028.616,296.743,373.033,170.890,46.441,158.972
C07184=1028.622,296.991,373.001,170.895,46.440,158.973
C07185=1028.629,297.238,372.968,170.899,46.440,158.973
C07186=1028.636,297.485,372.936,170.904,46.439,158.974
C07187=1028.643,297.734,372.903,170.909,46.439,158.974
C07188=1028.649,297.981,372.870,170.913,46.438,158.974
C07189=1028.655,298.229,372.837,170.917,46.437,158.975
C07190=1028.663,298.477,372.805,170.922,46.437,158.975
C07191=1028.669,298.724,372.772,170.927,46.436,158.976
C07192=1028.676,298.972,372.739,170.931,46.436,158.976
C07193=1028.683,299.220,372.707,170.935,46.436,158.976
C07194=1028.689,299.468,372.674,170.941,46.435,158.977
C07195=1028.696,299.716,372.641,170.945,46.435,158.977
C07196=1028.703,299.963,372.609,170.949,46.434,158.978
C07197=1028.710,300.211,372.576,170.954,46.434,158.978
C07198=1028.717,300.459,372.543,170.959,46.432,158.978
C07199=1028.724,300.706,372.510,170.963,46.432,158.979
C07200=1028.731,300.954,372.477,170.967,46.432,158.979
C07201=1028.737,301.202,372.444,170.972,46.431,158.980
C07202=1028.744,301.449,372.412,170.977,46.431,158.980
C07203=1028.751,301.697,372.379,170.981,46.430,158.981
C07204=1028.757,301.945,372.346,170.986,46.430,158.981
C07205=1028.765,302.192,372.313,170.991,46.429,158.981
C07206=1028.772,302.440,372.280,170.995,46.429,158.982
C07207=1028.778,302.688,372.247,171.000,46.428,158.982
C07208=1028.785,302.936,372.214,171.005,46.428,158.983
C07209=1028.793,303.183,372.181,171.010,46.428,158.983
C07210=1028.799,303.431,372.148,171.014,46.427,158.984
C07211=1028.806,303.679,372.115,171.019,46.427,158.984
C07212=1028.813,303.926,372.083,171.024,46.426,158.985
C07213=1028.820,304.174,372.049,171.028,46.426,158.985
C07214=1028.826,304.421,372.016,171.033,46.425,158.986
C07215=1028.834,304.669,371.983,171.038,46.425,158.986
C07216=1028.841,304.917,371.950,171.042,46.424,158.986
C07217=1028.847,305.165,371.917,171.047,46.424,158.987
C07218=1028.855,305.412,371.883,171.052,46.423,158.987
C07219=1028.862,305.660,371.851,171.056,46.424,158.988
C07220=1028.869,305.907,371.817,171.062,46.423,158.988
C07221=1028.880,306.326,371.762,171.069,46.422,158.989
C07222=1028.893,306.744,371.706,171.077,46.422,158.990
C07223=1028.904,307.163,371.650,171.086,46.421,158.991
C07224=1028.916,307.582,371.594,171.093,46.420,158.992
C07225=1028.923,307.828,371.561,171.099,46.420,158.992
C07226=1028.931,308.076,371.527,171.103,46.419,158.992
C07227=1028.937,308.324,371.494,171.107,46.419,158.993
C07228=1028.945,308.572,371.461,171.113,46.419,158.994
C07229=1028.952,308.819,371.428,171.117,46.418,158.994
C07230=1028.959,309.067,371.394,171.122,46.418,158.994
C07231=1028.966,309.315,371.360,171.127,46.418,158.995
C07232=1028.974,309.563,371.328,171.132,46.417,158.996
C07233=1028.980,309.810,371.294,171.137,46.417,158.996
C07234=1028.988,310.057,371.260,171.141,46.417,158.997
C07235=1028.995,310.305,371.227,171.147,46.416,158.997
C07236=1029.002,310.553,371.194,171.151,46.416,158.997
C07237=1029.009,310.800,371.161,171.157,46.416,158.998
C07238=1029.016,311.048,371.127,171.161,46.415,158.998
C07239=1029.023,311.295,371.093,171.167,46.415,158.999
C07240=1029.031,311.543,371.059,171.171,46.415,159.000
C07241=1029.036,311.790,371.025,171.176,46.415,159.000
C07242=1029.044,312.038,370.991,171.181,46.415,159.001
C07243=1029.051,312.286,370.957,171.185,46.415,159.001
C07244=1029.057,312.534,370.923,171.190,46.415,159.002
C07245=1029.064,312.780,370.890,171.196,46.415,159.002
C07246=1029.071,313.028,370.856,171.200,46.415,159.003
C07247=1029.078,313.276,370.821,171.206,46.414,159.004
C07248=1029.085,313.523,370.787,171.210,46.415,159.004
C07249=1029.091,313.770,370.753,171.215,46.414,159.005
C07250=1029.098,314.018,370.719,171.220,46.414,159.005
C07251=1029.105,314.266,370.685,171.225,46.414,159.006
C07252=1029.112,314.514,370.651,171.230,46.414,159.006
C07253=1029.119,314.761,370.616,171.235,46.414,159.007
C07254=1029.126,315.009,370.582,171.240,46.414,159.008
C07255=1029.132,315.256,370.548,171.245,46.414,159.008
C07256=1029.140,315.503,370.514,171.251,46.414,159.009
C07257=1029.147,315.751,370.480,171.255,46.414,159.009
C07258=1029.153,315.999,370.445,171.260,46.414,159.010
C07259=1029.161,316.246,370.412,171.265,46.414,159.010
C07260=1029.168,316.493,370.377,171.270,46.414,159.011
C07261=1029.175,316.741,370.343,171.275,46.414,159.012
C07262=1029.182,316.989,370.309,171.280,46.414,159.012
C07263=1029.189,317.236,370.274,171.286,46.414,159.013
C07264=1029.196,317.484,370.240,171.290,46.414,159.013
C07265=1029.203,317.732,370.206,171.296,46.414,159.014
C07266=1029.210,317.979,370.171,171.300,46.414,159.015
C07267=1029.217,318.227,370.137,171.306,46.414,159.015
C07268=1029.225,318.474,370.103,171.311,46.414,159.016
C07269=1029.231,318.722,370.068,171.316,46.414,159.016
C07270=1029.238,318.969,370.034,171.321,46.414,159.017
C07271=1029.245,319.217,369.999,171.326,46.414,159.018
C07272=1029.252,319.464,369.965,171.331,46.414,159.018
C07273=1029.260,319.711,369.931,171.337,46.414,159.019
C07274=1029.266,319.959,369.896,171.341,46.414,159.020
C07275=1029.274,320.206,369.861,171.347,46.414,159.020
C07276=1029.281,320.454,369.827,171.351,46.415,159.021
C07277=1029.287,320.665,369.798,171.356,46.415,159.021
C07278=1029.293,320.878,369.768,171.360,46.414,159.022
C07279=1029.300,321.089,369.738,171.365,46.415,159.022
C07280=1029.306,321.301,369.709,171.370,46.415,159.023
C07281=1029.311,321.512,369.679,171.374,46.415,159.024
